LIN {X 0,Y 250.03,Z 323.645,A -85,B 0,C 180,E1 -18844.205,E2 -18844.205} C_VEL
LIN {X 0,Y 249.102,Z 319.461,A -85,B 0,C 180,E1 -18845.837,E2 -18845.837} C_VEL
LIN {X 0,Y 249.003,Z 319.471,A -85,B 0,C 180,E1 -18850.477,E2 -18850.477} C_VEL
LIN {X 0,Y 248.982,Z 319.471,A -85,B 0,C 180,E1 -18854.882,E2 -18854.882} C_VEL
LIN {X 0,Y 249.005,Z 319.467,A -85,B 0,C 180,E1 -18857.361,E2 -18857.361} C_VEL
LIN {X 0,Y 249.035,Z 319.463,A -85,B 0,C 180,E1 -18861.621,E2 -18861.621} C_VEL
LIN {X 0,Y 249.057,Z 319.458,A -85,B 0,C 180,E1 -18865.642,E2 -18865.642} C_VEL
LIN {X 0,Y 249.047,Z 319.447,A -85,B 0,C 180,E1 -18869.473,E2 -18869.473} C_VEL
LIN {X 0,Y 249.068,Z 319.461,A -85,B 0,C 180,E1 -18873.162,E2 -18873.162} C_VEL
LIN {X 0,Y 249.074,Z 319.46,A -85,B 0,C 180,E1 -18876.732,E2 -18876.732} C_VEL
LIN {X 0,Y 249.105,Z 319.45,A -85,B 0,C 180,E1 -18880.211,E2 -18880.211} C_VEL
LIN {X 0,Y 249.237,Z 319.439,A -85,B 0,C 180,E1 -18883.622,E2 -18883.622} C_VEL
LIN {X 0,Y 249.248,Z 319.429,A -85,B 0,C 180,E1 -18888.617,E2 -18888.617} C_VEL
LIN {X 0,Y 249.477,Z 319.408,A -85,B 0,C 180,E1 -18891.903,E2 -18891.903} C_VEL
LIN {X 0,Y 249.43,Z 319.409,A -85,B 0,C 180,E1 -18896.77,E2 -18896.77} C_VEL
LIN {X 0,Y 249.722,Z 319.373,A -85,B 0,C 180,E1 -18900,E2 -18900} C_VEL
LIN {X 0,Y 249.427,Z 319.411,A -85,B 0,C 180,E1 -18903.231,E2 -18903.231} C_VEL
LIN {X 0,Y 249.428,Z 319.41,A -85,B 0,C 180,E1 -18906.549,E2 -18906.549} C_VEL
LIN {X 0,Y 249.339,Z 319.421,A -85,B 0,C 180,E1 -18909.737,E2 -18909.737} C_VEL
LIN {X 0,Y 249.201,Z 319.438,A -85,B 0,C 180,E1 -18914.704,E2 -18914.704} C_VEL
LIN {X 0,Y 249.134,Z 319.451,A -85,B 0,C 180,E1 -18918.078,E2 -18918.078} C_VEL
LIN {X 0,Y 249.079,Z 319.453,A -85,B 0,C 180,E1 -18921.519,E2 -18921.519} C_VEL
LIN {X 0,Y 249.081,Z 319.443,A -85,B 0,C 180,E1 -18925.461,E2 -18925.461} C_VEL
LIN {X 0,Y 249.035,Z 319.46,A -85,B 0,C 180,E1 -18928.976,E2 -18928.976} C_VEL
LIN {X 0,Y 249.024,Z 319.466,A -85,B 0,C 180,E1 -18932.427,E2 -18932.427} C_VEL
LIN {X 0,Y 249.044,Z 319.461,A -85,B 0,C 180,E1 -18936.344,E2 -18936.344} C_VEL
LIN {X 0,Y 249.004,Z 319.457,A -85,B 0,C 180,E1 -18940.479,E2 -18940.479} C_VEL
LIN {X 0,Y 248.984,Z 319.47,A -85,B 0,C 180,E1 -18944.884,E2 -18944.884} C_VEL
LIN {X 0,Y 249,Z 319.467,A -85,B 0,C 180,E1 -18947.361,E2 -18947.361} C_VEL
LIN {X 0,Y 249.041,Z 319.453,A -85,B 0,C 180,E1 -18952.202,E2 -18952.202} C_VEL
LIN {X 0,Y 249.043,Z 319.461,A -85,B 0,C 180,E1 -18955.641,E2 -18955.641} C_VEL
LIN {X 0,Y 249.002,Z 319.468,A -85,B 0,C 180,E1 -18959.468,E2 -18959.468} C_VEL
LIN {X 0,Y 249.036,Z 319.464,A -85,B 0,C 180,E1 -18963.159,E2 -18963.159} C_VEL
LIN {X 0,Y 249.055,Z 319.459,A -85,B 0,C 180,E1 -18966.731,E2 -18966.731} C_VEL
LIN {X 0,Y 249.088,Z 319.455,A -85,B 0,C 180,E1 -18970.211,E2 -18970.211} C_VEL
LIN {X 0,Y 249.198,Z 319.444,A -85,B 0,C 180,E1 -18973.62,E2 -18973.62} C_VEL
LIN {X 0,Y 249.245,Z 319.436,A -85,B 0,C 180,E1 -18978.617,E2 -18978.617} C_VEL
LIN {X 0,Y 249.438,Z 319.415,A -85,B 0,C 180,E1 -18981.902,E2 -18981.902} C_VEL
LIN {X 0,Y 249.255,Z 319.435,A -85,B 0,C 180,E1 -18985.149,E2 -18985.149} C_VEL
LIN {X 0,Y 249.65,Z 319.389,A -85,B 0,C 180,E1 -18988.388,E2 -18988.388} C_VEL
LIN {X 0,Y 249.649,Z 319.388,A -85,B 0,C 180,E1 -18991.614,E2 -18991.614} C_VEL
LIN {X 0,Y 249.424,Z 319.418,A -85,B 0,C 180,E1 -18996.472,E2 -18996.472} C_VEL
LIN {X 0,Y 249.335,Z 319.426,A -85,B 0,C 180,E1 -18999.738,E2 -18999.738} C_VEL
LIN {X 0,Y 249.146,Z 319.452,A -85,B 0,C 180,E1 -19004.708,E2 -19004.708} C_VEL
LIN {X 0,Y 249.137,Z 319.452,A -85,B 0,C 180,E1 -19007.325,E2 -19007.325} C_VEL
LIN {X 0,Y 250.767,Z 323.932,A -85,B 0,C 180,E1 -19007.655,E2 -19007.655} C_VEL
LIN {X 0,Y 258.308,Z 343.81,A -85,B 0,C 180,E1 -19009.057,E2 -19009.057} C_VEL
LIN {X 0,Y 262.117,Z 355.153,A -85,B 0,C 180,E1 -19009.774,E2 -19009.774} C_VEL
LIN {X 0,Y 259.34,Z 426.653,A -85,B 0,C 180,E1 -19012.022,E2 -19012.022} C_VEL
LIN {X 0,Y 258.384,Z 440.539,A -85,B 0,C 180,E1 -19012.778,E2 -19012.778} C_VEL
LIN {X 0,Y 257.341,Z 452.554,A -85,B 0,C 180,E1 -19013.731,E2 -19013.731} C_VEL
LIN {X 0,Y 255.946,Z 464.685,A -85,B 0,C 180,E1 -19015.02,E2 -19015.02} C_VEL
LIN {X 0,Y 254.367,Z 476.702,A -85,B 0,C 180,E1 -19016.671,E2 -19016.671} C_VEL
LIN {X 0,Y 252.928,Z 486.716,A -85,B 0,C 180,E1 -19018.415,E2 -19018.415} C_VEL
LIN {X 0,Y 251.406,Z 496.138,A -85,B 0,C 180,E1 -19020.444,E2 -19020.444} C_VEL
LIN {X 0,Y 250.107,Z 504.061,A -85,B 0,C 180,E1 -19022.541,E2 -19022.541} C_VEL
LIN {X 0,Y 248.917,Z 511.656,A -85,B 0,C 180,E1 -19025.034,E2 -19025.034} C_VEL
LIN {X 0,Y 248.031,Z 517.544,A -85,B 0,C 180,E1 -19027.496,E2 -19027.496} C_VEL
LIN {X 0,Y 247.458,Z 522.104,A -85,B 0,C 180,E1 -19029.93,E2 -19029.93} C_VEL
LIN {X 0,Y 246.793,Z 526.425,A -85,B 0,C 180,E1 -19033.115,E2 -19033.115} C_VEL
LIN {X 0,Y 246.614,Z 528.472,A -85,B 0,C 180,E1 -19035.435,E2 -19035.435} C_VEL
LIN {X 0,Y 246.681,Z 529.69,A -85,B 0,C 180,E1 -19037.796,E2 -19037.796} C_VEL
LIN {X 0,Y 246.872,Z 530.061,A -85,B 0,C 180,E1 -19040.233,E2 -19040.233} C_VEL
LIN {X 0,Y 247.505,Z 529.204,A -85,B 0,C 180,E1 -19043.394,E2 -19043.394} C_VEL
LIN {X 0,Y 248.58,Z 526.802,A -85,B 0,C 180,E1 -19046.542,E2 -19046.542} C_VEL
LIN {X 0,Y 250.07,Z 522.874,A -85,B 0,C 180,E1 -19049.61,E2 -19049.61} C_VEL
LIN {X 0,Y 251.955,Z 517.798,A -85,B 0,C 180,E1 -19052.381,E2 -19052.381} C_VEL
LIN {X 0,Y 254.299,Z 511.152,A -85,B 0,C 180,E1 -19055.073,E2 -19055.073} C_VEL
LIN {X 0,Y 256.78,Z 503.593,A -85,B 0,C 180,E1 -19057.469,E2 -19057.469} C_VEL
LIN {X 0,Y 259.517,Z 494.561,A -85,B 0,C 180,E1 -19059.713,E2 -19059.713} C_VEL
LIN {X 0,Y 262.243,Z 484.71,A -85,B 0,C 180,E1 -19061.645,E2 -19061.645} C_VEL
LIN {X 0,Y 264.805,Z 474.366,A -85,B 0,C 180,E1 -19063.258,E2 -19063.258} C_VEL
LIN {X 0,Y 267.225,Z 462.907,A -85,B 0,C 180,E1 -19064.654,E2 -19064.654} C_VEL
LIN {X 0,Y 269.363,Z 450.034,A -85,B 0,C 180,E1 -19065.862,E2 -19065.862} C_VEL
LIN {X 0,Y 270.921,Z 437.319,A -85,B 0,C 180,E1 -19066.734,E2 -19066.734} C_VEL
LIN {X 0,Y 272.145,Z 423.426,A -85,B 0,C 180,E1 -19067.343,E2 -19067.343} C_VEL
LIN {X 0,Y 275.677,Z 365.669,A -85,B 0,C 180,E1 -19069.121,E2 -19069.121} C_VEL
LIN {X 0,Y 270.019,Z 353.323,A -85,B 0,C 180,E1 -19070.753,E2 -19070.753} C_VEL
LIN {X 0,Y 263.673,Z 341.842,A -85,B 0,C 180,E1 -19072.672,E2 -19072.672} C_VEL
LIN {X 0,Y 259.384,Z 334.783,A -85,B 0,C 180,E1 -19074.07,E2 -19074.07} C_VEL
LIN {X 0,Y 256.653,Z 330.712,A -85,B 0,C 180,E1 -19074.992,E2 -19074.992} C_VEL
LIN {X 0,Y 250.933,Z 322.884,A -85,B 0,C 180,E1 -19077.065,E2 -19077.065} C_VEL
LIN {X 0,Y 249.681,Z 321.815,A -85,B 0,C 180,E1 -19077.526,E2 -19077.526} C_VEL
LIN {X 0,Y 248.305,Z 321.348,A -85,B 0,C 180,E1 -19078.029,E2 -19078.029} C_VEL
LIN {X 0,Y 244.436,Z 320.951,A -85,B 0,C 180,E1 -19079.7,E2 -19079.7} C_VEL
LIN {X 0,Y 242.856,Z 320.376,A -85,B 0,C 180,E1 -19080.934,E2 -19080.934} C_VEL
LIN {X 0,Y 242.635,Z 320.256,A -85,B 0,C 180,E1 -19081.579,E2 -19081.579} C_VEL
LIN {X 0,Y 242.411,Z 320.281,A -85,B 0,C 180,E1 -19086.659,E2 -19086.659} C_VEL
LIN {X 0,Y 242.27,Z 320.297,A -85,B 0,C 180,E1 -19090.023,E2 -19090.023} C_VEL
LIN {X 0,Y 242.139,Z 320.323,A -85,B 0,C 180,E1 -19095.142,E2 -19095.142} C_VEL
LIN {X 0,Y 242.052,Z 320.331,A -85,B 0,C 180,E1 -19098.625,E2 -19098.625} C_VEL
LIN {X 0,Y 242.007,Z 320.335,A -85,B 0,C 180,E1 -19102.18,E2 -19102.18} C_VEL
LIN {X 0,Y 242.069,Z 320.328,A -85,B 0,C 180,E1 -19105.838,E2 -19105.838} C_VEL
LIN {X 0,Y 242.031,Z 320.336,A -85,B 0,C 180,E1 -19109.58,E2 -19109.58} C_VEL
LIN {X 0,Y 241.983,Z 320.342,A -85,B 0,C 180,E1 -19113.492,E2 -19113.492} C_VEL
LIN {X 0,Y 241.991,Z 320.335,A -85,B 0,C 180,E1 -19117.581,E2 -19117.581} C_VEL
LIN {X 0,Y 241.971,Z 320.532,A -85,B 0,C 180,E1 -19121.083,E2 -19121.083} C_VEL
LIN {X 0,Y 243.323,Z 324.398,A -85,B 0,C 180,E1 -19123.884,E2 -19123.884} C_VEL
LIN {X 0,Y 245.036,Z 329.254,A -85,B 0,C 180,E1 -19127.001,E2 -19127.001} C_VEL
LIN {X 0,Y 245.857,Z 331.663,A -85,B 0,C 180,E1 -19128.294,E2 -19128.294} C_VEL
LIN {X 0,Y 249.084,Z 336.698,A -85,B 0,C 180,E1 -19129.624,E2 -19129.624} C_VEL
LIN {X 0,Y 253.954,Z 344.732,A -85,B 0,C 180,E1 -19131.478,E2 -19131.478} C_VEL
LIN {X 0,Y 257.084,Z 350.374,A -85,B 0,C 180,E1 -19132.593,E2 -19132.593} C_VEL
LIN {X 0,Y 261.696,Z 359.399,A -85,B 0,C 180,E1 -19134.165,E2 -19134.165} C_VEL
LIN {X 0,Y 266.799,Z 370.947,A -85,B 0,C 180,E1 -19135.818,E2 -19135.818} C_VEL
LIN {X 0,Y 268.746,Z 386.31,A -85,B 0,C 180,E1 -19136.893,E2 -19136.893} C_VEL
LIN {X 0,Y 269.128,Z 390.539,A -85,B 0,C 180,E1 -19137.149,E2 -19137.149} C_VEL
LIN {X 0,Y 265.736,Z 443.432,A -85,B 0,C 180,E1 -19138.843,E2 -19138.843} C_VEL
LIN {X 0,Y 264.156,Z 456.738,A -85,B 0,C 180,E1 -19139.524,E2 -19139.524} C_VEL
LIN {X 0,Y 261.95,Z 469.593,A -85,B 0,C 180,E1 -19140.462,E2 -19140.462} C_VEL
LIN {X 0,Y 259.418,Z 481.764,A -85,B 0,C 180,E1 -19141.698,E2 -19141.698} C_VEL
LIN {X 0,Y 256.562,Z 492.835,A -85,B 0,C 180,E1 -19143.128,E2 -19143.128} C_VEL
LIN {X 0,Y 253.881,Z 502.949,A -85,B 0,C 180,E1 -19144.81,E2 -19144.81} C_VEL
LIN {X 0,Y 251.337,Z 511.329,A -85,B 0,C 180,E1 -19146.517,E2 -19146.517} C_VEL
LIN {X 0,Y 248.356,Z 520.484,A -85,B 0,C 180,E1 -19148.85,E2 -19148.85} C_VEL
LIN {X 0,Y 245.962,Z 527.909,A -85,B 0,C 180,E1 -19151.248,E2 -19151.248} C_VEL
LIN {X 0,Y 243.566,Z 534.796,A -85,B 0,C 180,E1 -19154.09,E2 -19154.09} C_VEL
LIN {X 0,Y 241.883,Z 539.395,A -85,B 0,C 180,E1 -19156.558,E2 -19156.558} C_VEL
LIN {X 0,Y 240.875,Z 542.931,A -85,B 0,C 180,E1 -19159.067,E2 -19159.067} C_VEL
LIN {X 0,Y 240.207,Z 545.478,A -85,B 0,C 180,E1 -19161.587,E2 -19161.587} C_VEL
LIN {X 0,Y 239.84,Z 547.387,A -85,B 0,C 180,E1 -19164.956,E2 -19164.956} C_VEL
LIN {X 0,Y 239.816,Z 547.753,A -85,B 0,C 180,E1 -19166.639,E2 -19166.639} C_VEL
LIN {X 0,Y 239.905,Z 547.721,A -85,B 0,C 180,E1 -19168.32,E2 -19168.32} C_VEL
LIN {X 0,Y 239.958,Z 547.237,A -85,B 0,C 180,E1 -19169.999,E2 -19169.999} C_VEL
LIN {X 0,Y 239.945,Z 546.336,A -85,B 0,C 180,E1 -19171.677,E2 -19171.677} C_VEL
LIN {X 0,Y 239.905,Z 545.015,A -85,B 0,C 180,E1 -19173.358,E2 -19173.358} C_VEL
LIN {X 0,Y 239.916,Z 542.156,A -85,B 0,C 180,E1 -19175.883,E2 -19175.883} C_VEL
LIN {X 0,Y 240.201,Z 538.208,A -85,B 0,C 180,E1 -19178.411,E2 -19178.411} C_VEL
LIN {X 0,Y 240.846,Z 532.063,A -85,B 0,C 180,E1 -19181.359,E2 -19181.359} C_VEL
LIN {X 0,Y 241.813,Z 525.276,A -85,B 0,C 180,E1 -19183.872,E2 -19183.872} C_VEL
LIN {X 0,Y 243.178,Z 516.827,A -85,B 0,C 180,E1 -19186.365,E2 -19186.365} C_VEL
LIN {X 0,Y 244.719,Z 507.213,A -85,B 0,C 180,E1 -19188.61,E2 -19188.61} C_VEL
LIN {X 0,Y 246.198,Z 497.332,A -85,B 0,C 180,E1 -19190.467,E2 -19190.467} C_VEL
LIN {X 0,Y 247.876,Z 486.712,A -85,B 0,C 180,E1 -19192.065,E2 -19192.065} C_VEL
LIN {X 0,Y 249.528,Z 474.972,A -85,B 0,C 180,E1 -19193.442,E2 -19193.442} C_VEL
LIN {X 0,Y 250.995,Z 461.662,A -85,B 0,C 180,E1 -19194.613,E2 -19194.613} C_VEL
LIN {X 0,Y 252.092,Z 449.229,A -85,B 0,C 180,E1 -19195.38,E2 -19195.38} C_VEL
LIN {X 0,Y 252.828,Z 433.94,A -85,B 0,C 180,E1 -19195.963,E2 -19195.963} C_VEL
LIN {X 0,Y 254.548,Z 385.732,A -85,B 0,C 180,E1 -19197.51,E2 -19197.51} C_VEL
LIN {X 0,Y 249.883,Z 349.342,A -85,B 0,C 180,E1 -19199.23,E2 -19199.23} C_VEL
LIN {X 0,Y 245.337,Z 336.056,A -85,B 0,C 180,E1 -19200.196,E2 -19200.196} C_VEL
LIN {X 0,Y 243.169,Z 325.344,A -85,B 0,C 180,E1 -19204.302,E2 -19204.302} C_VEL
LIN {X 0,Y 242.085,Z 320.336,A -85,B 0,C 180,E1 -19206.34,E2 -19206.34} C_VEL
LIN {X 0,Y 241.928,Z 320.349,A -85,B 0,C 180,E1 -19210.949,E2 -19210.949} C_VEL
LIN {X 0,Y 241.915,Z 320.352,A -85,B 0,C 180,E1 -19214.204,E2 -19214.204} C_VEL
LIN {X 0,Y 241.935,Z 320.349,A -85,B 0,C 180,E1 -19218.077,E2 -19218.077} C_VEL
LIN {X 0,Y 241.999,Z 320.342,A -85,B 0,C 180,E1 -19222.42,E2 -19222.42} C_VEL
LIN {X 0,Y 241.987,Z 320.341,A -85,B 0,C 180,E1 -19226.509,E2 -19226.509} C_VEL
LIN {X 0,Y 242.032,Z 320.322,A -85,B 0,C 180,E1 -19230.587,E2 -19230.587} C_VEL
LIN {X 0,Y 242.063,Z 320.331,A -85,B 0,C 180,E1 -19234.183,E2 -19234.183} C_VEL
LIN {X 0,Y 242.048,Z 320.331,A -85,B 0,C 180,E1 -19238.297,E2 -19238.297} C_VEL
LIN {X 0,Y 242.158,Z 320.323,A -85,B 0,C 180,E1 -19243.278,E2 -19243.278} C_VEL
LIN {X 0,Y 242.181,Z 320.309,A -85,B 0,C 180,E1 -19248.28,E2 -19248.28} C_VEL
LIN {X 0,Y 242.423,Z 320.288,A -85,B 0,C 180,E1 -19251.666,E2 -19251.666} C_VEL
LIN {X 0,Y 242.254,Z 320.306,A -85,B 0,C 180,E1 -19255.007,E2 -19255.007} C_VEL
LIN {X 0,Y 242.631,Z 320.251,A -85,B 0,C 180,E1 -19258.341,E2 -19258.341} C_VEL
LIN {X 0,Y 242.63,Z 320.257,A -85,B 0,C 180,E1 -19261.66,E2 -19261.66} C_VEL
LIN {X 0,Y 242.404,Z 320.285,A -85,B 0,C 180,E1 -19266.66,E2 -19266.66} C_VEL
LIN {X 0,Y 242.263,Z 320.298,A -85,B 0,C 180,E1 -19270.024,E2 -19270.024} C_VEL
LIN {X 0,Y 242.163,Z 320.313,A -85,B 0,C 180,E1 -19275.142,E2 -19275.142} C_VEL
LIN {X 0,Y 242.068,Z 320.329,A -85,B 0,C 180,E1 -19278.625,E2 -19278.625} C_VEL
LIN {X 0,Y 242.001,Z 320.336,A -85,B 0,C 180,E1 -19282.182,E2 -19282.182} C_VEL
LIN {X 0,Y 242.029,Z 320.321,A -85,B 0,C 180,E1 -19285.822,E2 -19285.822} C_VEL
LIN {X 0,Y 241.966,Z 320.339,A -85,B 0,C 180,E1 -19289.589,E2 -19289.589} C_VEL
LIN {X 0,Y 241.976,Z 320.341,A -85,B 0,C 180,E1 -19293.494,E2 -19293.494} C_VEL
LIN {X 0,Y 241.986,Z 320.334,A -85,B 0,C 180,E1 -19297.583,E2 -19297.583} C_VEL
LIN {X 0,Y 241.931,Z 320.34,A -85,B 0,C 180,E1 -19301.924,E2 -19301.924} C_VEL
LIN {X 0,Y 241.919,Z 320.349,A -85,B 0,C 180,E1 -19306.576,E2 -19306.576} C_VEL
LIN {X 0,Y 241.992,Z 320.332,A -85,B 0,C 180,E1 -19311.642,E2 -19311.642} C_VEL
LIN {X 0,Y 241.986,Z 320.335,A -85,B 0,C 180,E1 -19314.491,E2 -19314.491} C_VEL
LIN {X 0,Y 241.953,Z 320.344,A -85,B 0,C 180,E1 -19318.478,E2 -19318.478} C_VEL
LIN {X 0,Y 241.968,Z 320.342,A -85,B 0,C 180,E1 -19322.309,E2 -19322.309} C_VEL
LIN {X 0,Y 242.026,Z 320.336,A -85,B 0,C 180,E1 -19326.014,E2 -19326.014} C_VEL
LIN {X 0,Y 242.023,Z 320.338,A -85,B 0,C 180,E1 -19329.608,E2 -19329.608} C_VEL
LIN {X 0,Y 242.118,Z 320.324,A -85,B 0,C 180,E1 -19333.317,E2 -19333.317} C_VEL
LIN {X 0,Y 242.156,Z 320.318,A -85,B 0,C 180,E1 -19336.576,E2 -19336.576} C_VEL
LIN {X 0,Y 242.388,Z 320.291,A -85,B 0,C 180,E1 -19341.665,E2 -19341.665} C_VEL
LIN {X 0,Y 242.403,Z 320.289,A -85,B 0,C 180,E1 -19343.341,E2 -19343.341} C_VEL
LIN {X 0,Y 242.609,Z 320.266,A -85,B 0,C 180,E1 -19348.341,E2 -19348.341} C_VEL
LIN {X 0,Y 242.609,Z 320.265,A -85,B 0,C 180,E1 -19351.661,E2 -19351.661} C_VEL
LIN {X 0,Y 242.394,Z 320.293,A -85,B 0,C 180,E1 -19356.661,E2 -19356.661} C_VEL
LIN {X 0,Y 242.263,Z 320.308,A -85,B 0,C 180,E1 -19360.025,E2 -19360.025} C_VEL
LIN {X 0,Y 242.105,Z 320.329,A -85,B 0,C 180,E1 -19365.146,E2 -19365.146} C_VEL
LIN {X 0,Y 242.124,Z 320.327,A -85,B 0,C 180,E1 -19366.651,E2 -19366.651} C_VEL
LIN {X 0,Y 243.549,Z 324.322,A -85,B 0,C 180,E1 -19366.962,E2 -19366.962} C_VEL
LIN {X 0,Y 248.831,Z 337.497,A -85,B 0,C 180,E1 -19367.96,E2 -19367.96} C_VEL
LIN {X 0,Y 255.38,Z 356.241,A -85,B 0,C 180,E1 -19369.232,E2 -19369.232} C_VEL
LIN {X 0,Y 252.609,Z 426.976,A -85,B 0,C 180,E1 -19371.525,E2 -19371.525} C_VEL
LIN {X 0,Y 251.648,Z 440.232,A -85,B 0,C 180,E1 -19372.258,E2 -19372.258} C_VEL
LIN {X 0,Y 250.597,Z 452.306,A -85,B 0,C 180,E1 -19373.228,E2 -19373.228} C_VEL
LIN {X 0,Y 249.119,Z 464.887,A -85,B 0,C 180,E1 -19374.591,E2 -19374.591} C_VEL
LIN {X 0,Y 247.486,Z 476.854,A -85,B 0,C 180,E1 -19376.274,E2 -19376.274} C_VEL
LIN {X 0,Y 245.91,Z 487.572,A -85,B 0,C 180,E1 -19378.203,E2 -19378.203} C_VEL
LIN {X 0,Y 244.314,Z 497.132,A -85,B 0,C 180,E1 -19380.345,E2 -19380.345} C_VEL
LIN {X 0,Y 243.082,Z 504.382,A -85,B 0,C 180,E1 -19382.336,E2 -19382.336} C_VEL
LIN {X 0,Y 241.834,Z 512.047,A -85,B 0,C 180,E1 -19384.933,E2 -19384.933} C_VEL
LIN {X 0,Y 240.877,Z 518.544,A -85,B 0,C 180,E1 -19387.787,E2 -19387.787} C_VEL
LIN {X 0,Y 240.219,Z 523.22,A -85,B 0,C 180,E1 -19390.476,E2 -19390.476} C_VEL
LIN {X 0,Y 239.73,Z 526.314,A -85,B 0,C 180,E1 -19392.868,E2 -19392.868} C_VEL
LIN {X 0,Y 239.532,Z 528.483,A -85,B 0,C 180,E1 -19395.236,E2 -19395.236} C_VEL
LIN {X 0,Y 239.591,Z 529.814,A -85,B 0,C 180,E1 -19397.571,E2 -19397.571} C_VEL
LIN {X 0,Y 239.748,Z 530.34,A -85,B 0,C 180,E1 -19399.84,E2 -19399.84} C_VEL
LIN {X 0,Y 240.119,Z 530.09,A -85,B 0,C 180,E1 -19402.211,E2 -19402.211} C_VEL
LIN {X 0,Y 240.827,Z 528.903,A -85,B 0,C 180,E1 -19404.798,E2 -19404.798} C_VEL
LIN {X 0,Y 241.866,Z 526.68,A -85,B 0,C 180,E1 -19407.424,E2 -19407.424} C_VEL
LIN {X 0,Y 243.251,Z 523.312,A -85,B 0,C 180,E1 -19410.085,E2 -19410.085} C_VEL
LIN {X 0,Y 245.101,Z 518.698,A -85,B 0,C 180,E1 -19412.735,E2 -19412.735} C_VEL
LIN {X 0,Y 247.418,Z 512.645,A -85,B 0,C 180,E1 -19415.365,E2 -19415.365} C_VEL
LIN {X 0,Y 250.163,Z 504.78,A -85,B 0,C 180,E1 -19417.987,E2 -19417.987} C_VEL
LIN {X 0,Y 253.136,Z 495.698,A -85,B 0,C 180,E1 -19420.349,E2 -19420.349} C_VEL
LIN {X 0,Y 255.77,Z 486.696,A -85,B 0,C 180,E1 -19422.2,E2 -19422.2} C_VEL
LIN {X 0,Y 258.828,Z 475.208,A -85,B 0,C 180,E1 -19424.072,E2 -19424.072} C_VEL
LIN {X 0,Y 261.347,Z 464.019,A -85,B 0,C 180,E1 -19425.49,E2 -19425.49} C_VEL
LIN {X 0,Y 263.611,Z 451.481,A -85,B 0,C 180,E1 -19426.706,E2 -19426.706} C_VEL
LIN {X 0,Y 265.308,Z 438.816,A -85,B 0,C 180,E1 -19427.619,E2 -19427.619} C_VEL
LIN {X 0,Y 266.587,Z 425.001,A -85,B 0,C 180,E1 -19428.264,E2 -19428.264} C_VEL
LIN {X 0,Y 270.177,Z 367.755,A -85,B 0,C 180,E1 -19430.076,E2 -19430.076} C_VEL
LIN {X 0,Y 264.553,Z 355.604,A -85,B 0,C 180,E1 -19431.817,E2 -19431.817} C_VEL
LIN {X 0,Y 258.185,Z 344.023,A -85,B 0,C 180,E1 -19433.896,E2 -19433.896} C_VEL
LIN {X 0,Y 253.236,Z 336.294,A -85,B 0,C 180,E1 -19435.617,E2 -19435.617} C_VEL
LIN {X 0,Y 245.251,Z 324.921,A -85,B 0,C 180,E1 -19438.773,E2 -19438.773} C_VEL
LIN {X 0,Y 243.331,Z 322.513,A -85,B 0,C 180,E1 -19439.601,E2 -19439.601} C_VEL
LIN {X 0,Y 243.054,Z 321.797,A -85,B 0,C 180,E1 -19439.772,E2 -19439.772} C_VEL
LIN {X 0,Y 242.628,Z 320.256,A -85,B 0,C 180,E1 -19440.933,E2 -19440.933} C_VEL
LIN {X 0,Y 242.635,Z 320.256,A -85,B 0,C 180,E1 -19441.579,E2 -19441.579} C_VEL
LIN {X 0,Y 242.34,Z 320.299,A -85,B 0,C 180,E1 -19442.504,E2 -19442.504} C_VEL
LIN {X 0,Y 240.983,Z 320.474,A -85,B 0,C 180,E1 -19443.867,E2 -19443.867} C_VEL
LIN {X 0,Y 236.525,Z 321.032,A -85,B 0,C 180,E1 -19447.045,E2 -19447.045} C_VEL
LIN {X 0,Y 235.408,Z 321.162,A -85,B 0,C 180,E1 -19448.471,E2 -19448.471} C_VEL
LIN {X 0,Y 235.303,Z 321.171,A -85,B 0,C 180,E1 -19448.955,E2 -19448.955} C_VEL
LIN {X 0,Y 235.093,Z 321.19,A -85,B 0,C 180,E1 -19453.836,E2 -19453.836} C_VEL
LIN {X 0,Y 235.021,Z 321.199,A -85,B 0,C 180,E1 -19457.399,E2 -19457.399} C_VEL
LIN {X 0,Y 234.978,Z 321.209,A -85,B 0,C 180,E1 -19461.998,E2 -19461.998} C_VEL
LIN {X 0,Y 234.971,Z 321.212,A -85,B 0,C 180,E1 -19466.657,E2 -19466.657} C_VEL
LIN {X 0,Y 234.933,Z 321.214,A -85,B 0,C 180,E1 -19470.567,E2 -19470.567} C_VEL
LIN {X 0,Y 234.932,Z 321.212,A -85,B 0,C 180,E1 -19474.637,E2 -19474.637} C_VEL
LIN {X 0,Y 234.969,Z 321.317,A -85,B 0,C 180,E1 -19478.226,E2 -19478.226} C_VEL
LIN {X 0,Y 237.053,Z 327.105,A -85,B 0,C 180,E1 -19482.991,E2 -19482.991} C_VEL
LIN {X 0,Y 238.301,Z 330.865,A -85,B 0,C 180,E1 -19485.507,E2 -19485.507} C_VEL
LIN {X 0,Y 242.379,Z 336.87,A -85,B 0,C 180,E1 -19487.449,E2 -19487.449} C_VEL
LIN {X 0,Y 246.9,Z 344.12,A -85,B 0,C 180,E1 -19489.396,E2 -19489.396} C_VEL
LIN {X 0,Y 251,Z 351.189,A -85,B 0,C 180,E1 -19491.025,E2 -19491.025} C_VEL
LIN {X 0,Y 255.403,Z 359.563,A -85,B 0,C 180,E1 -19492.644,E2 -19492.644} C_VEL
LIN {X 0,Y 260,Z 369.572,A -85,B 0,C 180,E1 -19494.269,E2 -19494.269} C_VEL
LIN {X 0,Y 262.019,Z 374.909,A -85,B 0,C 180,E1 -19494.975,E2 -19494.975} C_VEL
LIN {X 0,Y 263.585,Z 388.526,A -85,B 0,C 180,E1 -19495.949,E2 -19495.949} C_VEL
LIN {X 0,Y 263.739,Z 393.029,A -85,B 0,C 180,E1 -19496.189,E2 -19496.189} C_VEL
LIN {X 0,Y 260.34,Z 443.254,A -85,B 0,C 180,E1 -19497.837,E2 -19497.837} C_VEL
LIN {X 0,Y 258.671,Z 456.525,A -85,B 0,C 180,E1 -19498.521,E2 -19498.521} C_VEL
LIN {X 0,Y 256.509,Z 468.848,A -85,B 0,C 180,E1 -19499.429,E2 -19499.429} C_VEL
LIN {X 0,Y 254.017,Z 480.361,A -85,B 0,C 180,E1 -19500.586,E2 -19500.586} C_VEL
LIN {X 0,Y 250.689,Z 492.897,A -85,B 0,C 180,E1 -19502.219,E2 -19502.219} C_VEL
LIN {X 0,Y 247.835,Z 502.895,A -85,B 0,C 180,E1 -19503.924,E2 -19503.924} C_VEL
LIN {X 0,Y 244.893,Z 512.008,A -85,B 0,C 180,E1 -19505.86,E2 -19505.86} C_VEL
LIN {X 0,Y 241.738,Z 521.119,A -85,B 0,C 180,E1 -19508.287,E2 -19508.287} C_VEL
LIN {X 0,Y 239.245,Z 528.295,A -85,B 0,C 180,E1 -19510.708,E2 -19510.708} C_VEL
LIN {X 0,Y 236.739,Z 534.99,A -85,B 0,C 180,E1 -19513.618,E2 -19513.618} C_VEL
LIN {X 0,Y 234.955,Z 539.477,A -85,B 0,C 180,E1 -19516.154,E2 -19516.154} C_VEL
LIN {X 0,Y 234.222,Z 541.87,A -85,B 0,C 180,E1 -19517.874,E2 -19517.874} C_VEL
LIN {X 0,Y 233.597,Z 543.84,A -85,B 0,C 180,E1 -19519.599,E2 -19519.599} C_VEL
LIN {X 0,Y 233.177,Z 545.357,A -85,B 0,C 180,E1 -19521.331,E2 -19521.331} C_VEL
LIN {X 0,Y 232.743,Z 547.179,A -85,B 0,C 180,E1 -19524.802,E2 -19524.802} C_VEL
LIN {X 0,Y 232.72,Z 547.503,A -85,B 0,C 180,E1 -19526.536,E2 -19526.536} C_VEL
LIN {X 0,Y 232.812,Z 547.391,A -85,B 0,C 180,E1 -19528.269,E2 -19528.269} C_VEL
LIN {X 0,Y 232.888,Z 546.858,A -85,B 0,C 180,E1 -19529.999,E2 -19529.999} C_VEL
LIN {X 0,Y 232.876,Z 545.913,A -85,B 0,C 180,E1 -19531.728,E2 -19531.728} C_VEL
LIN {X 0,Y 232.807,Z 544.544,A -85,B 0,C 180,E1 -19533.46,E2 -19533.46} C_VEL
LIN {X 0,Y 232.855,Z 541.599,A -85,B 0,C 180,E1 -19536.063,E2 -19536.063} C_VEL
LIN {X 0,Y 233.164,Z 537.556,A -85,B 0,C 180,E1 -19538.667,E2 -19538.667} C_VEL
LIN {X 0,Y 233.845,Z 531.257,A -85,B 0,C 180,E1 -19541.703,E2 -19541.703} C_VEL
LIN {X 0,Y 234.899,Z 524.358,A -85,B 0,C 180,E1 -19544.289,E2 -19544.289} C_VEL
LIN {X 0,Y 236.351,Z 515.734,A -85,B 0,C 180,E1 -19546.852,E2 -19546.852} C_VEL
LIN {X 0,Y 237.811,Z 506.82,A -85,B 0,C 180,E1 -19548.969,E2 -19548.969} C_VEL
LIN {X 0,Y 239.529,Z 495.851,A -85,B 0,C 180,E1 -19551.064,E2 -19551.064} C_VEL
LIN {X 0,Y 241.193,Z 484.865,A -85,B 0,C 180,E1 -19552.71,E2 -19552.71} C_VEL
LIN {X 0,Y 243.037,Z 472.734,A -85,B 0,C 180,E1 -19554.107,E2 -19554.107} C_VEL
LIN {X 0,Y 244.252,Z 461.383,A -85,B 0,C 180,E1 -19555.112,E2 -19555.112} C_VEL
LIN {X 0,Y 245.372,Z 448.971,A -85,B 0,C 180,E1 -19555.898,E2 -19555.898} C_VEL
LIN {X 0,Y 246.121,Z 433.789,A -85,B 0,C 180,E1 -19556.497,E2 -19556.497} C_VEL
LIN {X 0,Y 247.891,Z 386.332,A -85,B 0,C 180,E1 -19558.064,E2 -19558.064} C_VEL
LIN {X 0,Y 243.343,Z 351.084,A -85,B 0,C 180,E1 -19559.777,E2 -19559.777} C_VEL
LIN {X 0,Y 238.08,Z 335.915,A -85,B 0,C 180,E1 -19560.89,E2 -19560.89} C_VEL
LIN {X 0,Y 235.955,Z 325.599,A -85,B 0,C 180,E1 -19564.984,E2 -19564.984} C_VEL
LIN {X 0,Y 234.998,Z 321.218,A -85,B 0,C 180,E1 -19566.868,E2 -19566.868} C_VEL
LIN {X 0,Y 234.877,Z 321.227,A -85,B 0,C 180,E1 -19571.578,E2 -19571.578} C_VEL
LIN {X 0,Y 234.88,Z 321.226,A -85,B 0,C 180,E1 -19575.898,E2 -19575.898} C_VEL
LIN {X 0,Y 234.891,Z 321.228,A -85,B 0,C 180,E1 -19578.834,E2 -19578.834} C_VEL
LIN {X 0,Y 234.951,Z 321.219,A -85,B 0,C 180,E1 -19581.085,E2 -19581.085} C_VEL
LIN {X 0,Y 234.956,Z 321.216,A -85,B 0,C 180,E1 -19585.367,E2 -19585.367} C_VEL
LIN {X 0,Y 234.965,Z 321.199,A -85,B 0,C 180,E1 -19590.157,E2 -19590.157} C_VEL
LIN {X 0,Y 234.989,Z 321.212,A -85,B 0,C 180,E1 -19593.793,E2 -19593.793} C_VEL
LIN {X 0,Y 235.007,Z 321.21,A -85,B 0,C 180,E1 -19598.97,E2 -19598.97} C_VEL
LIN {X 0,Y 235.092,Z 321.202,A -85,B 0,C 180,E1 -19603.059,E2 -19603.059} C_VEL
LIN {X 0,Y 235.142,Z 321.186,A -85,B 0,C 180,E1 -19607.924,E2 -19607.924} C_VEL
LIN {X 0,Y 235.372,Z 321.165,A -85,B 0,C 180,E1 -19611.414,E2 -19611.414} C_VEL
LIN {X 0,Y 235.399,Z 321.162,A -85,B 0,C 180,E1 -19613.142,E2 -19613.142} C_VEL
LIN {X 0,Y 235.591,Z 321.127,A -85,B 0,C 180,E1 -19618.291,E2 -19618.291} C_VEL
LIN {X 0,Y 235.59,Z 321.134,A -85,B 0,C 180,E1 -19621.71,E2 -19621.71} C_VEL
LIN {X 0,Y 235.355,Z 321.163,A -85,B 0,C 180,E1 -19626.861,E2 -19626.861} C_VEL
LIN {X 0,Y 235.21,Z 321.174,A -85,B 0,C 180,E1 -19630.328,E2 -19630.328} C_VEL
LIN {X 0,Y 235.11,Z 321.192,A -85,B 0,C 180,E1 -19635.607,E2 -19635.607} C_VEL
LIN {X 0,Y 235.003,Z 321.207,A -85,B 0,C 180,E1 -19639.207,E2 -19639.207} C_VEL
LIN {X 0,Y 234.943,Z 321.21,A -85,B 0,C 180,E1 -19642.885,E2 -19642.885} C_VEL
LIN {X 0,Y 234.942,Z 321.209,A -85,B 0,C 180,E1 -19646.661,E2 -19646.661} C_VEL
LIN {X 0,Y 234.896,Z 321.225,A -85,B 0,C 180,E1 -19650.574,E2 -19650.574} C_VEL
LIN {X 0,Y 234.927,Z 321.222,A -85,B 0,C 180,E1 -19654.639,E2 -19654.639} C_VEL
LIN {X 0,Y 234.94,Z 321.208,A -85,B 0,C 180,E1 -19658.946,E2 -19658.946} C_VEL
LIN {X 0,Y 234.876,Z 321.224,A -85,B 0,C 180,E1 -19663.489,E2 -19663.489} C_VEL
LIN {X 0,Y 234.872,Z 321.227,A -85,B 0,C 180,E1 -19666.512,E2 -19666.512} C_VEL
LIN {X 0,Y 234.917,Z 321.217,A -85,B 0,C 180,E1 -19671.08,E2 -19671.08} C_VEL
LIN {X 0,Y 234.929,Z 321.22,A -85,B 0,C 180,E1 -19675.363,E2 -19675.363} C_VEL
LIN {X 0,Y 234.899,Z 321.225,A -85,B 0,C 180,E1 -19679.429,E2 -19679.429} C_VEL
LIN {X 0,Y 234.97,Z 321.215,A -85,B 0,C 180,E1 -19683.808,E2 -19683.808} C_VEL
LIN {X 0,Y 234.991,Z 321.211,A -85,B 0,C 180,E1 -19688.969,E2 -19688.969} C_VEL
LIN {X 0,Y 235.058,Z 321.203,A -85,B 0,C 180,E1 -19693.093,E2 -19693.093} C_VEL
LIN {X 0,Y 235.112,Z 321.199,A -85,B 0,C 180,E1 -19697.923,E2 -19697.923} C_VEL
LIN {X 0,Y 235.322,Z 321.17,A -85,B 0,C 180,E1 -19701.413,E2 -19701.413} C_VEL
LIN {X 0,Y 235.355,Z 321.166,A -85,B 0,C 180,E1 -19703.141,E2 -19703.141} C_VEL
LIN {X 0,Y 235.568,Z 321.144,A -85,B 0,C 180,E1 -19708.291,E2 -19708.291} C_VEL
LIN {X 0,Y 235.567,Z 321.143,A -85,B 0,C 180,E1 -19711.711,E2 -19711.711} C_VEL
LIN {X 0,Y 235.345,Z 321.17,A -85,B 0,C 180,E1 -19716.861,E2 -19716.861} C_VEL
LIN {X 0,Y 235.187,Z 321.19,A -85,B 0,C 180,E1 -19720.33,E2 -19720.33} C_VEL
LIN {X 0,Y 235.046,Z 321.208,A -85,B 0,C 180,E1 -19725.612,E2 -19725.612} C_VEL
LIN {X 0,Y 235.085,Z 321.322,A -85,B 0,C 180,E1 -19725.976,E2 -19725.976} C_VEL
LIN {X 0,Y 236.012,Z 323.987,A -85,B 0,C 180,E1 -19726.178,E2 -19726.178} C_VEL
LIN {X 0,Y 241.767,Z 337.895,A -85,B 0,C 180,E1 -19727.302,E2 -19727.302} C_VEL
LIN {X 0,Y 248.803,Z 357.945,A -85,B 0,C 180,E1 -19728.705,E2 -19728.705} C_VEL
LIN {X 0,Y 245.905,Z 427.111,A -85,B 0,C 180,E1 -19731.006,E2 -19731.006} C_VEL
LIN {X 0,Y 244.849,Z 441.043,A -85,B 0,C 180,E1 -19731.802,E2 -19731.802} C_VEL
LIN {X 0,Y 243.834,Z 452.214,A -85,B 0,C 180,E1 -19732.728,E2 -19732.728} C_VEL
LIN {X 0,Y 242.405,Z 464.365,A -85,B 0,C 180,E1 -19734.061,E2 -19734.061} C_VEL
LIN {X 0,Y 240.687,Z 476.602,A -85,B 0,C 180,E1 -19735.81,E2 -19735.81} C_VEL
LIN {X 0,Y 239.049,Z 487.356,A -85,B 0,C 180,E1 -19737.774,E2 -19737.774} C_VEL
LIN {X 0,Y 237.38,Z 496.992,A -85,B 0,C 180,E1 -19739.975,E2 -19739.975} C_VEL
LIN {X 0,Y 235.89,Z 505.637,A -85,B 0,C 180,E1 -19742.432,E2 -19742.432} C_VEL
LIN {X 0,Y 234.517,Z 513.512,A -85,B 0,C 180,E1 -19745.295,E2 -19745.295} C_VEL
LIN {X 0,Y 233.795,Z 518.78,A -85,B 0,C 180,E1 -19747.723,E2 -19747.723} C_VEL
LIN {X 0,Y 233.207,Z 522.911,A -85,B 0,C 180,E1 -19750.122,E2 -19750.122} C_VEL
LIN {X 0,Y 232.554,Z 527.161,A -85,B 0,C 180,E1 -19753.505,E2 -19753.505} C_VEL
LIN {X 0,Y 232.425,Z 529.479,A -85,B 0,C 180,E1 -19756.528,E2 -19756.528} C_VEL
LIN {X 0,Y 232.564,Z 530.476,A -85,B 0,C 180,E1 -19759.069,E2 -19759.069} C_VEL
LIN {X 0,Y 232.929,Z 530.577,A -85,B 0,C 180,E1 -19761.674,E2 -19761.674} C_VEL
LIN {X 0,Y 233.846,Z 529.244,A -85,B 0,C 180,E1 -19765.177,E2 -19765.177} C_VEL
LIN {X 0,Y 235.258,Z 526.464,A -85,B 0,C 180,E1 -19768.48,E2 -19768.48} C_VEL
LIN {X 0,Y 237.18,Z 522.092,A -85,B 0,C 180,E1 -19771.698,E2 -19771.698} C_VEL
LIN {X 0,Y 239.485,Z 516.619,A -85,B 0,C 180,E1 -19774.574,E2 -19774.574} C_VEL
LIN {X 0,Y 241.78,Z 510.871,A -85,B 0,C 180,E1 -19776.895,E2 -19776.895} C_VEL
LIN {X 0,Y 244.659,Z 503.069,A -85,B 0,C 180,E1 -19779.396,E2 -19779.396} C_VEL
LIN {X 0,Y 247.466,Z 494.778,A -85,B 0,C 180,E1 -19781.502,E2 -19781.502} C_VEL
LIN {X 0,Y 250.475,Z 484.962,A -85,B 0,C 180,E1 -19783.492,E2 -19783.492} C_VEL
LIN {X 0,Y 253.253,Z 474.805,A -85,B 0,C 180,E1 -19785.126,E2 -19785.126} C_VEL
LIN {X 0,Y 256.085,Z 462.818,A -85,B 0,C 180,E1 -19786.611,E2 -19786.611} C_VEL
LIN {X 0,Y 258.355,Z 450.27,A -85,B 0,C 180,E1 -19787.817,E2 -19787.817} C_VEL
LIN {X 0,Y 259.922,Z 438.382,A -85,B 0,C 180,E1 -19788.662,E2 -19788.662} C_VEL
LIN {X 0,Y 261.24,Z 425.13,A -85,B 0,C 180,E1 -19789.277,E2 -19789.277} C_VEL
LIN {X 0,Y 264.907,Z 370.247,A -85,B 0,C 180,E1 -19791.056,E2 -19791.056} C_VEL
LIN {X 0,Y 260.153,Z 359.919,A -85,B 0,C 180,E1 -19792.603,E2 -19792.603} C_VEL
LIN {X 0,Y 254.092,Z 348.637,A -85,B 0,C 180,E1 -19794.712,E2 -19794.712} C_VEL
LIN {X 0,Y 249.96,Z 341.936,A -85,B 0,C 180,E1 -19796.241,E2 -19796.241} C_VEL
LIN {X 0,Y 242.379,Z 330.944,A -85,B 0,C 180,E1 -19799.377,E2 -19799.377} C_VEL
LIN {X 0,Y 240.251,Z 328.032,A -85,B 0,C 180,E1 -19800.367,E2 -19800.367} C_VEL
LIN {X 0,Y 238.343,Z 325.916,A -85,B 0,C 180,E1 -19801.267,E2 -19801.267} C_VEL
LIN {X 0,Y 236.113,Z 323.353,A -85,B 0,C 180,E1 -19802.399,E2 -19802.399} C_VEL
LIN {X 0,Y 235.647,Z 322.348,A -85,B 0,C 180,E1 -19802.778,E2 -19802.778} C_VEL
LIN {X 0,Y 235.263,Z 321.172,A -85,B 0,C 180,E1 -19803.854,E2 -19803.854} C_VEL
LIN {X 0,Y 235.363,Z 321.158,A -85,B 0,C 180,E1 -19806.859,E2 -19806.859} C_VEL
LIN {X 0,Y 235.303,Z 321.171,A -85,B 0,C 180,E1 -19808.955,E2 -19808.955} C_VEL
LIN {X 0,Y 234.583,Z 321.256,A -85,B 0,C 180,E1 -19810.382,E2 -19810.382} C_VEL
LIN {X 0,Y 231.657,Z 321.622,A -85,B 0,C 180,E1 -19812.706,E2 -19812.706} C_VEL
LIN {X 0,Y 229.18,Z 321.934,A -85,B 0,C 180,E1 -19814.601,E2 -19814.601} C_VEL
LIN {X 0,Y 228.101,Z 322.068,A -85,B 0,C 180,E1 -19816.074,E2 -19816.074} C_VEL
LIN {X 0,Y 228.002,Z 322.075,A -85,B 0,C 180,E1 -19816.574,E2 -19816.574} C_VEL
LIN {X 0,Y 227.947,Z 322.082,A -85,B 0,C 180,E1 -19821.714,E2 -19821.714} C_VEL
LIN {X 0,Y 227.945,Z 322.088,A -85,B 0,C 180,E1 -19826.602,E2 -19826.602} C_VEL
LIN {X 0,Y 227.91,Z 322.091,A -85,B 0,C 180,E1 -19830.295,E2 -19830.295} C_VEL
LIN {X 0,Y 227.898,Z 322.168,A -85,B 0,C 180,E1 -19834.517,E2 -19834.517} C_VEL
LIN {X 0,Y 229.077,Z 325.158,A -85,B 0,C 180,E1 -19837.85,E2 -19837.85} C_VEL
LIN {X 0,Y 230.715,Z 330.063,A -85,B 0,C 180,E1 -19842.079,E2 -19842.079} C_VEL
LIN {X 0,Y 234.996,Z 336.176,A -85,B 0,C 180,E1 -19844.557,E2 -19844.557} C_VEL
LIN {X 0,Y 239.999,Z 343.745,A -85,B 0,C 180,E1 -19847.061,E2 -19847.061} C_VEL
LIN {X 0,Y 243.731,Z 349.894,A -85,B 0,C 180,E1 -19848.746,E2 -19848.746} C_VEL
LIN {X 0,Y 248.293,Z 357.926,A -85,B 0,C 180,E1 -19850.63,E2 -19850.63} C_VEL
LIN {X 0,Y 253.824,Z 369.422,A -85,B 0,C 180,E1 -19852.757,E2 -19852.757} C_VEL
LIN {X 0,Y 257.169,Z 377.775,A -85,B 0,C 180,E1 -19854.016,E2 -19854.016} C_VEL
LIN {X 0,Y 258.64,Z 391.733,A -85,B 0,C 180,E1 -19855.027,E2 -19855.027} C_VEL
LIN {X 0,Y 255.511,Z 438.357,A -85,B 0,C 180,E1 -19856.584,E2 -19856.584} C_VEL
LIN {X 0,Y 253.952,Z 452.343,A -85,B 0,C 180,E1 -19857.221,E2 -19857.221} C_VEL
LIN {X 0,Y 251.569,Z 466.083,A -85,B 0,C 180,E1 -19858.176,E2 -19858.176} C_VEL
LIN {X 0,Y 249.121,Z 477.307,A -85,B 0,C 180,E1 -19859.247,E2 -19859.247} C_VEL
LIN {X 0,Y 246.044,Z 489.13,A -85,B 0,C 180,E1 -19860.714,E2 -19860.714} C_VEL
LIN {X 0,Y 243.518,Z 497.62,A -85,B 0,C 180,E1 -19862.031,E2 -19862.031} C_VEL
LIN {X 0,Y 240.196,Z 507.646,A -85,B 0,C 180,E1 -19863.966,E2 -19863.966} C_VEL
LIN {X 0,Y 236.793,Z 517.397,A -85,B 0,C 180,E1 -19866.378,E2 -19866.378} C_VEL
LIN {X 0,Y 233.742,Z 525.29,A -85,B 0,C 180,E1 -19868.849,E2 -19868.849} C_VEL
LIN {X 0,Y 231.395,Z 531.641,A -85,B 0,C 180,E1 -19871.402,E2 -19871.402} C_VEL
LIN {X 0,Y 229.24,Z 536.78,A -85,B 0,C 180,E1 -19873.982,E2 -19873.982} C_VEL
LIN {X 0,Y 227.622,Z 540.799,A -85,B 0,C 180,E1 -19876.61,E2 -19876.61} C_VEL
LIN {X 0,Y 226.592,Z 543.8,A -85,B 0,C 180,E1 -19879.274,E2 -19879.274} C_VEL
LIN {X 0,Y 225.808,Z 546.305,A -85,B 0,C 180,E1 -19882.847,E2 -19882.847} C_VEL
LIN {X 0,Y 225.638,Z 547.108,A -85,B 0,C 180,E1 -19885.352,E2 -19885.352} C_VEL
LIN {X 0,Y 225.722,Z 547.055,A -85,B 0,C 180,E1 -19888.215,E2 -19888.215} C_VEL
LIN {X 0,Y 225.819,Z 546.48,A -85,B 0,C 180,E1 -19889.999,E2 -19889.999} C_VEL
LIN {X 0,Y 225.785,Z 545.49,A -85,B 0,C 180,E1 -19891.783,E2 -19891.783} C_VEL
LIN {X 0,Y 225.758,Z 542.538,A -85,B 0,C 180,E1 -19895.009,E2 -19895.009} C_VEL
LIN {X 0,Y 225.992,Z 538.348,A -85,B 0,C 180,E1 -19898.043,E2 -19898.043} C_VEL
LIN {X 0,Y 226.483,Z 533.389,A -85,B 0,C 180,E1 -19900.729,E2 -19900.729} C_VEL
LIN {X 0,Y 227.331,Z 527.095,A -85,B 0,C 180,E1 -19903.406,E2 -19903.406} C_VEL
LIN {X 0,Y 228.633,Z 519.212,A -85,B 0,C 180,E1 -19906.059,E2 -19906.059} C_VEL
LIN {X 0,Y 229.971,Z 511.681,A -85,B 0,C 180,E1 -19908.112,E2 -19908.112} C_VEL
LIN {X 0,Y 231.772,Z 501.242,A -85,B 0,C 180,E1 -19910.407,E2 -19910.407} C_VEL
LIN {X 0,Y 233.323,Z 491.579,A -85,B 0,C 180,E1 -19912.117,E2 -19912.117} C_VEL
LIN {X 0,Y 234.94,Z 481.272,A -85,B 0,C 180,E1 -19913.583,E2 -19913.583} C_VEL
LIN {X 0,Y 236.579,Z 469.085,A -85,B 0,C 180,E1 -19914.926,E2 -19914.926} C_VEL
LIN {X 0,Y 238.04,Z 455.859,A -85,B 0,C 180,E1 -19915.991,E2 -19915.991} C_VEL
LIN {X 0,Y 239.008,Z 442.81,A -85,B 0,C 180,E1 -19916.7,E2 -19916.7} C_VEL
LIN {X 0,Y 241.222,Z 386.695,A -85,B 0,C 180,E1 -19918.631,E2 -19918.631} C_VEL
LIN {X 0,Y 236.918,Z 353.232,A -85,B 0,C 180,E1 -19920.316,E2 -19920.316} C_VEL
LIN {X 0,Y 230.767,Z 335.634,A -85,B 0,C 180,E1 -19921.673,E2 -19921.673} C_VEL
LIN {X 0,Y 228.764,Z 325.813,A -85,B 0,C 180,E1 -19925.71,E2 -19925.71} C_VEL
LIN {X 0,Y 227.941,Z 322.097,A -85,B 0,C 180,E1 -19927.326,E2 -19927.326} C_VEL
LIN {X 0,Y 227.804,Z 322.11,A -85,B 0,C 180,E1 -19932.233,E2 -19932.233} C_VEL
LIN {X 0,Y 227.822,Z 322.105,A -85,B 0,C 180,E1 -19935.194,E2 -19935.194} C_VEL
LIN {X 0,Y 227.828,Z 322.105,A -85,B 0,C 180,E1 -19939.624,E2 -19939.624} C_VEL
LIN {X 0,Y 227.896,Z 322.096,A -85,B 0,C 180,E1 -19944.131,E2 -19944.131} C_VEL
LIN {X 0,Y 227.868,Z 322.091,A -85,B 0,C 180,E1 -19948.378,E2 -19948.378} C_VEL
LIN {X 0,Y 227.881,Z 322.093,A -85,B 0,C 180,E1 -19952.445,E2 -19952.445} C_VEL
LIN {X 0,Y 227.91,Z 322.096,A -85,B 0,C 180,E1 -19956.367,E2 -19956.367} C_VEL
LIN {X 0,Y 227.938,Z 322.086,A -85,B 0,C 180,E1 -19960.174,E2 -19960.174} C_VEL
LIN {X 0,Y 228.053,Z 322.077,A -85,B 0,C 180,E1 -19963.898,E2 -19963.898} C_VEL
LIN {X 0,Y 228.089,Z 322.066,A -85,B 0,C 180,E1 -19967.544,E2 -19967.544} C_VEL
LIN {X 0,Y 228.301,Z 322.044,A -85,B 0,C 180,E1 -19971.146,E2 -19971.146} C_VEL
LIN {X 0,Y 228.35,Z 322.039,A -85,B 0,C 180,E1 -19972.929,E2 -19972.929} C_VEL
LIN {X 0,Y 228.549,Z 322.004,A -85,B 0,C 180,E1 -19978.238,E2 -19978.238} C_VEL
LIN {X 0,Y 228.548,Z 322.011,A -85,B 0,C 180,E1 -19981.763,E2 -19981.763} C_VEL
LIN {X 0,Y 228.307,Z 322.041,A -85,B 0,C 180,E1 -19987.073,E2 -19987.073} C_VEL
LIN {X 0,Y 228.141,Z 322.052,A -85,B 0,C 180,E1 -19990.652,E2 -19990.652} C_VEL
LIN {X 0,Y 228.061,Z 322.07,A -85,B 0,C 180,E1 -19994.273,E2 -19994.273} C_VEL
LIN {X 0,Y 227.999,Z 322.082,A -85,B 0,C 180,E1 -19997.954,E2 -19997.954} C_VEL
LIN {X 0,Y 227.917,Z 322.088,A -85,B 0,C 180,E1 -20002.325,E2 -20002.325} C_VEL
LIN {X 0,Y 227.919,Z 322.082,A -85,B 0,C 180,E1 -20006.593,E2 -20006.593} C_VEL
LIN {X 0,Y 227.87,Z 322.097,A -85,B 0,C 180,E1 -20010.282,E2 -20010.282} C_VEL
LIN {X 0,Y 227.874,Z 322.098,A -85,B 0,C 180,E1 -20013.722,E2 -20013.722} C_VEL
LIN {X 0,Y 227.841,Z 322.096,A -85,B 0,C 180,E1 -20018.092,E2 -20018.092} C_VEL
LIN {X 0,Y 227.804,Z 322.103,A -85,B 0,C 180,E1 -20022.745,E2 -20022.745} C_VEL
LIN {X 0,Y 227.798,Z 322.109,A -85,B 0,C 180,E1 -20027.256,E2 -20027.256} C_VEL
LIN {X 0,Y 227.843,Z 322.092,A -85,B 0,C 180,E1 -20031.91,E2 -20031.91} C_VEL
LIN {X 0,Y 227.879,Z 322.096,A -85,B 0,C 180,E1 -20036.379,E2 -20036.379} C_VEL
LIN {X 0,Y 227.877,Z 322.096,A -85,B 0,C 180,E1 -20040.433,E2 -20040.433} C_VEL
LIN {X 0,Y 227.903,Z 322.094,A -85,B 0,C 180,E1 -20044.424,E2 -20044.424} C_VEL
LIN {X 0,Y 227.953,Z 322.088,A -85,B 0,C 180,E1 -20048.287,E2 -20048.287} C_VEL
LIN {X 0,Y 228.026,Z 322.081,A -85,B 0,C 180,E1 -20053.897,E2 -20053.897} C_VEL
LIN {X 0,Y 228.069,Z 322.075,A -85,B 0,C 180,E1 -20057.544,E2 -20057.544} C_VEL
LIN {X 0,Y 228.26,Z 322.048,A -85,B 0,C 180,E1 -20061.145,E2 -20061.145} C_VEL
LIN {X 0,Y 228.308,Z 322.044,A -85,B 0,C 180,E1 -20062.928,E2 -20062.928} C_VEL
LIN {X 0,Y 228.502,Z 322.025,A -85,B 0,C 180,E1 -20068.239,E2 -20068.239} C_VEL
LIN {X 0,Y 228.501,Z 322.023,A -85,B 0,C 180,E1 -20071.764,E2 -20071.764} C_VEL
LIN {X 0,Y 228.297,Z 322.047,A -85,B 0,C 180,E1 -20077.074,E2 -20077.074} C_VEL
LIN {X 0,Y 228.127,Z 322.07,A -85,B 0,C 180,E1 -20080.653,E2 -20080.653} C_VEL
LIN {X 0,Y 227.998,Z 322.087,A -85,B 0,C 180,E1 -20085.19,E2 -20085.19} C_VEL
LIN {X 0,Y 229.147,Z 325.168,A -85,B 0,C 180,E1 -20085.482,E2 -20085.482} C_VEL
LIN {X 0,Y 235.235,Z 339.73,A -85,B 0,C 180,E1 -20086.713,E2 -20086.713} C_VEL
LIN {X 0,Y 242.068,Z 359.17,A -85,B 0,C 180,E1 -20088.134,E2 -20088.134} C_VEL
LIN {X 0,Y 239.148,Z 427.76,A -85,B 0,C 180,E1 -20090.494,E2 -20090.494} C_VEL
LIN {X 0,Y 238.072,Z 441.593,A -85,B 0,C 180,E1 -20091.314,E2 -20091.314} C_VEL
LIN {X 0,Y 236.941,Z 453.432,A -85,B 0,C 180,E1 -20092.337,E2 -20092.337} C_VEL
LIN {X 0,Y 235.364,Z 466.108,A -85,B 0,C 180,E1 -20093.809,E2 -20093.809} C_VEL
LIN {X 0,Y 233.664,Z 477.629,A -85,B 0,C 180,E1 -20095.533,E2 -20095.533} C_VEL
LIN {X 0,Y 231.946,Z 488.511,A -85,B 0,C 180,E1 -20097.621,E2 -20097.621} C_VEL
LIN {X 0,Y 230.183,Z 498.431,A -85,B 0,C 180,E1 -20099.999,E2 -20099.999} C_VEL
LIN {X 0,Y 228.713,Z 506.805,A -85,B 0,C 180,E1 -20102.531,E2 -20102.531} C_VEL
LIN {X 0,Y 227.355,Z 514.373,A -85,B 0,C 180,E1 -20105.423,E2 -20105.423} C_VEL
LIN {X 0,Y 226.532,Z 520.314,A -85,B 0,C 180,E1 -20108.353,E2 -20108.353} C_VEL
LIN {X 0,Y 225.912,Z 524.127,A -85,B 0,C 180,E1 -20110.792,E2 -20110.792} C_VEL
LIN {X 0,Y 225.388,Z 527.913,A -85,B 0,C 180,E1 -20114.177,E2 -20114.177} C_VEL
LIN {X 0,Y 225.327,Z 529.715,A -85,B 0,C 180,E1 -20116.67,E2 -20116.67} C_VEL
LIN {X 0,Y 225.471,Z 530.688,A -85,B 0,C 180,E1 -20119.112,E2 -20119.112} C_VEL
LIN {X 0,Y 225.798,Z 530.891,A -85,B 0,C 180,E1 -20121.5,E2 -20121.5} C_VEL
LIN {X 0,Y 226.339,Z 530.421,A -85,B 0,C 180,E1 -20123.845,E2 -20123.845} C_VEL
LIN {X 0,Y 227.273,Z 528.949,A -85,B 0,C 180,E1 -20126.609,E2 -20126.609} C_VEL
LIN {X 0,Y 228.61,Z 526.405,A -85,B 0,C 180,E1 -20129.406,E2 -20129.406} C_VEL
LIN {X 0,Y 230.393,Z 522.683,A -85,B 0,C 180,E1 -20132.207,E2 -20132.207} C_VEL
LIN {X 0,Y 232.671,Z 517.68,A -85,B 0,C 180,E1 -20134.983,E2 -20134.983} C_VEL
LIN {X 0,Y 235.457,Z 511.227,A -85,B 0,C 180,E1 -20137.715,E2 -20137.715} C_VEL
LIN {X 0,Y 238.019,Z 504.724,A -85,B 0,C 180,E1 -20139.893,E2 -20139.893} C_VEL
LIN {X 0,Y 241.13,Z 496.204,A -85,B 0,C 180,E1 -20142.18,E2 -20142.18} C_VEL
LIN {X 0,Y 244.148,Z 487.028,A -85,B 0,C 180,E1 -20144.129,E2 -20144.129} C_VEL
LIN {X 0,Y 247.06,Z 477.117,A -85,B 0,C 180,E1 -20145.813,E2 -20145.813} C_VEL
LIN {X 0,Y 249.948,Z 465.855,A -85,B 0,C 180,E1 -20147.332,E2 -20147.332} C_VEL
LIN {X 0,Y 252.382,Z 454.117,A -85,B 0,C 180,E1 -20148.549,E2 -20148.549} C_VEL
LIN {X 0,Y 254.329,Z 441.475,A -85,B 0,C 180,E1 -20149.539,E2 -20149.539} C_VEL
LIN {X 0,Y 255.805,Z 429.148,A -85,B 0,C 180,E1 -20150.188,E2 -20150.188} C_VEL
LIN {X 0,Y 259.716,Z 372.727,A -85,B 0,C 180,E1 -20152.081,E2 -20152.081} C_VEL
LIN {X 0,Y 255.732,Z 363.967,A -85,B 0,C 180,E1 -20153.48,E2 -20153.48} C_VEL
LIN {X 0,Y 250.214,Z 353.498,A -85,B 0,C 180,E1 -20155.502,E2 -20155.502} C_VEL
LIN {X 0,Y 246.082,Z 346.749,A -85,B 0,C 180,E1 -20157.135,E2 -20157.135} C_VEL
LIN {X 0,Y 239.567,Z 336.945,A -85,B 0,C 180,E1 -20160,E2 -20160} C_VEL
LIN {X 0,Y 236.428,Z 332.671,A -85,B 0,C 180,E1 -20161.54,E2 -20161.54} C_VEL
LIN {X 0,Y 233.713,Z 329.699,A -85,B 0,C 180,E1 -20162.962,E2 -20162.962} C_VEL
LIN {X 0,Y 232.414,Z 327.942,A -85,B 0,C 180,E1 -20163.711,E2 -20163.711} C_VEL
LIN {X 0,Y 229.477,Z 325.311,A -85,B 0,C 180,E1 -20165.437,E2 -20165.437} C_VEL
LIN {X 0,Y 228.477,Z 323.131,A -85,B 0,C 180,E1 -20166.291,E2 -20166.291} C_VEL
LIN {X 0,Y 228.279,Z 322.041,A -85,B 0,C 180,E1 -20167.518,E2 -20167.518} C_VEL
LIN {X 0,Y 228.148,Z 322.057,A -85,B 0,C 180,E1 -20170.651,E2 -20170.651} C_VEL
LIN {X 0,Y 228.048,Z 322.069,A -85,B 0,C 180,E1 -20174.273,E2 -20174.273} C_VEL
LIN {X 0,Y 228.002,Z 322.075,A -85,B 0,C 180,E1 -20176.574,E2 -20176.574} C_VEL
LIN {X 0,Y 227.31,Z 322.164,A -85,B 0,C 180,E1 -20178.046,E2 -20178.046} C_VEL
LIN {X 0,Y 224.464,Z 322.514,A -85,B 0,C 180,E1 -20180.449,E2 -20180.449} C_VEL
LIN {X 0,Y 221.213,Z 322.923,A -85,B 0,C 180,E1 -20183.418,E2 -20183.418} C_VEL
LIN {X 0,Y 220.864,Z 322.961,A -85,B 0,C 180,E1 -20184.446,E2 -20184.446} C_VEL
LIN {X 0,Y 220.826,Z 322.967,A -85,B 0,C 180,E1 -20188.644,E2 -20188.644} C_VEL
LIN {X 0,Y 222.247,Z 326.64,A -85,B 0,C 180,E1 -20194.695,E2 -20194.695} C_VEL
LIN {X 0,Y 223.365,Z 329.335,A -85,B 0,C 180,E1 -20197.681,E2 -20197.681} C_VEL
LIN {X 0,Y 226.36,Z 333.98,A -85,B 0,C 180,E1 -20200.096,E2 -20200.096} C_VEL
LIN {X 0,Y 228.854,Z 337.088,A -85,B 0,C 180,E1 -20201.76,E2 -20201.76} C_VEL
LIN {X 0,Y 233.395,Z 343.757,A -85,B 0,C 180,E1 -20204.457,E2 -20204.457} C_VEL
LIN {X 0,Y 237.241,Z 349.887,A -85,B 0,C 180,E1 -20206.46,E2 -20206.46} C_VEL
LIN {X 0,Y 240.437,Z 355.319,A -85,B 0,C 180,E1 -20207.99,E2 -20207.99} C_VEL
LIN {X 0,Y 244.782,Z 363.264,A -85,B 0,C 180,E1 -20209.89,E2 -20209.89} C_VEL
LIN {X 0,Y 250.064,Z 374.706,A -85,B 0,C 180,E1 -20212.057,E2 -20212.057} C_VEL
LIN {X 0,Y 252.538,Z 381.217,A -85,B 0,C 180,E1 -20213.049,E2 -20213.049} C_VEL
LIN {X 0,Y 253.623,Z 393.142,A -85,B 0,C 180,E1 -20213.942,E2 -20213.942} C_VEL
LIN {X 0,Y 249.966,Z 443.052,A -85,B 0,C 180,E1 -20215.662,E2 -20215.662} C_VEL
LIN {X 0,Y 248.14,Z 456.098,A -85,B 0,C 180,E1 -20216.353,E2 -20216.353} C_VEL
LIN {X 0,Y 245.665,Z 468.794,A -85,B 0,C 180,E1 -20217.317,E2 -20217.317} C_VEL
LIN {X 0,Y 242.763,Z 480.89,A -85,B 0,C 180,E1 -20218.593,E2 -20218.593} C_VEL
LIN {X 0,Y 239.578,Z 491.896,A -85,B 0,C 180,E1 -20220.086,E2 -20220.086} C_VEL
LIN {X 0,Y 236.319,Z 501.951,A -85,B 0,C 180,E1 -20221.827,E2 -20221.827} C_VEL
LIN {X 0,Y 232.704,Z 511.91,A -85,B 0,C 180,E1 -20224.028,E2 -20224.028} C_VEL
LIN {X 0,Y 229.216,Z 520.8,A -85,B 0,C 180,E1 -20226.509,E2 -20226.509} C_VEL
LIN {X 0,Y 226.04,Z 528.533,A -85,B 0,C 180,E1 -20229.3,E2 -20229.3} C_VEL
LIN {X 0,Y 223.904,Z 533.775,A -85,B 0,C 180,E1 -20231.706,E2 -20231.706} C_VEL
LIN {X 0,Y 221.753,Z 538.389,A -85,B 0,C 180,E1 -20234.371,E2 -20234.371} C_VEL
LIN {X 0,Y 220.299,Z 541.94,A -85,B 0,C 180,E1 -20237.095,E2 -20237.095} C_VEL
LIN {X 0,Y 219.087,Z 545.145,A -85,B 0,C 180,E1 -20240.769,E2 -20240.769} C_VEL
LIN {X 0,Y 218.735,Z 546.154,A -85,B 0,C 180,E1 -20242.615,E2 -20242.615} C_VEL
LIN {X 0,Y 218.547,Z 546.897,A -85,B 0,C 180,E1 -20245.48,E2 -20245.48} C_VEL
LIN {X 0,Y 218.634,Z 546.712,A -85,B 0,C 180,E1 -20248.157,E2 -20248.157} C_VEL
LIN {X 0,Y 218.751,Z 546.095,A -85,B 0,C 180,E1 -20249.999,E2 -20249.999} C_VEL
LIN {X 0,Y 218.695,Z 545.047,A -85,B 0,C 180,E1 -20251.84,E2 -20251.84} C_VEL
LIN {X 0,Y 218.693,Z 542.199,A -85,B 0,C 180,E1 -20254.978,E2 -20254.978} C_VEL
LIN {X 0,Y 218.927,Z 537.679,A -85,B 0,C 180,E1 -20258.305,E2 -20258.305} C_VEL
LIN {X 0,Y 219.47,Z 532.61,A -85,B 0,C 180,E1 -20261.076,E2 -20261.076} C_VEL
LIN {X 0,Y 220.398,Z 526.191,A -85,B 0,C 180,E1 -20263.836,E2 -20263.836} C_VEL
LIN {X 0,Y 221.755,Z 518.099,A -85,B 0,C 180,E1 -20266.572,E2 -20266.572} C_VEL
LIN {X 0,Y 223.14,Z 510.137,A -85,B 0,C 180,E1 -20268.751,E2 -20268.751} C_VEL
LIN {X 0,Y 225.071,Z 499.758,A -85,B 0,C 180,E1 -20271.043,E2 -20271.043} C_VEL
LIN {X 0,Y 226.741,Z 489.825,A -85,B 0,C 180,E1 -20272.794,E2 -20272.794} C_VEL
LIN {X 0,Y 228.369,Z 479.078,A -85,B 0,C 180,E1 -20274.305,E2 -20274.305} C_VEL
LIN {X 0,Y 229.961,Z 467.432,A -85,B 0,C 180,E1 -20275.573,E2 -20275.573} C_VEL
LIN {X 0,Y 231.399,Z 454.49,A -85,B 0,C 180,E1 -20276.613,E2 -20276.613} C_VEL
LIN {X 0,Y 232.335,Z 441.905,A -85,B 0,C 180,E1 -20277.287,E2 -20277.287} C_VEL
LIN {X 0,Y 234.548,Z 387.085,A -85,B 0,C 180,E1 -20279.227,E2 -20279.227} C_VEL
LIN {X 0,Y 230.579,Z 355.596,A -85,B 0,C 180,E1 -20280.87,E2 -20280.87} C_VEL
LIN {X 0,Y 223.484,Z 335.362,A -85,B 0,C 180,E1 -20282.487,E2 -20282.487} C_VEL
LIN {X 0,Y 221.572,Z 325.997,A -85,B 0,C 180,E1 -20286.491,E2 -20286.491} C_VEL
LIN {X 0,Y 220.895,Z 322.974,A -85,B 0,C 180,E1 -20287.909,E2 -20287.909} C_VEL
LIN {X 0,Y 220.758,Z 322.987,A -85,B 0,C 180,E1 -20292.927,E2 -20292.927} C_VEL
LIN {X 0,Y 220.76,Z 322.987,A -85,B 0,C 180,E1 -20297.071,E2 -20297.071} C_VEL
LIN {X 0,Y 220.805,Z 322.982,A -85,B 0,C 180,E1 -20300.463,E2 -20300.463} C_VEL
LIN {X 0,Y 220.828,Z 322.978,A -85,B 0,C 180,E1 -20302.794,E2 -20302.794} C_VEL
LIN {X 0,Y 220.82,Z 322.971,A -85,B 0,C 180,E1 -20307.245,E2 -20307.245} C_VEL
LIN {X 0,Y 220.832,Z 322.971,A -85,B 0,C 180,E1 -20311.486,E2 -20311.486} C_VEL
LIN {X 0,Y 220.863,Z 322.974,A -85,B 0,C 180,E1 -20315.565,E2 -20315.565} C_VEL
LIN {X 0,Y 220.888,Z 322.966,A -85,B 0,C 180,E1 -20319.514,E2 -20319.514} C_VEL
LIN {X 0,Y 221.012,Z 322.957,A -85,B 0,C 180,E1 -20323.37,E2 -20323.37} C_VEL
LIN {X 0,Y 221.107,Z 322.934,A -85,B 0,C 180,E1 -20329.006,E2 -20329.006} C_VEL
LIN {X 0,Y 221.285,Z 322.918,A -85,B 0,C 180,E1 -20332.702,E2 -20332.702} C_VEL
LIN {X 0,Y 221.507,Z 322.881,A -85,B 0,C 180,E1 -20338.182,E2 -20338.182} C_VEL
LIN {X 0,Y 221.506,Z 322.889,A -85,B 0,C 180,E1 -20341.819,E2 -20341.819} C_VEL
LIN {X 0,Y 221.243,Z 322.921,A -85,B 0,C 180,E1 -20347.3,E2 -20347.3} C_VEL
LIN {X 0,Y 221.063,Z 322.932,A -85,B 0,C 180,E1 -20350.997,E2 -20350.997} C_VEL
LIN {X 0,Y 220.992,Z 322.95,A -85,B 0,C 180,E1 -20354.74,E2 -20354.74} C_VEL
LIN {X 0,Y 220.916,Z 322.964,A -85,B 0,C 180,E1 -20358.55,E2 -20358.55} C_VEL
LIN {X 0,Y 220.864,Z 322.963,A -85,B 0,C 180,E1 -20362.666,E2 -20362.666} C_VEL
LIN {X 0,Y 220.862,Z 322.963,A -85,B 0,C 180,E1 -20367.006,E2 -20367.006} C_VEL
LIN {X 0,Y 220.815,Z 322.979,A -85,B 0,C 180,E1 -20370.76,E2 -20370.76} C_VEL
LIN {X 0,Y 220.798,Z 322.979,A -85,B 0,C 180,E1 -20374.956,E2 -20374.956} C_VEL
LIN {X 0,Y 220.804,Z 322.964,A -85,B 0,C 180,E1 -20379.538,E2 -20379.538} C_VEL
LIN {X 0,Y 220.765,Z 322.982,A -85,B 0,C 180,E1 -20384.457,E2 -20384.457} C_VEL
LIN {X 0,Y 220.757,Z 322.984,A -85,B 0,C 180,E1 -20388.046,E2 -20388.046} C_VEL
LIN {X 0,Y 220.824,Z 322.967,A -85,B 0,C 180,E1 -20392.794,E2 -20392.794} C_VEL
LIN {X 0,Y 220.812,Z 322.98,A -85,B 0,C 180,E1 -20397.245,E2 -20397.245} C_VEL
LIN {X 0,Y 220.805,Z 322.981,A -85,B 0,C 180,E1 -20401.483,E2 -20401.483} C_VEL
LIN {X 0,Y 220.848,Z 322.975,A -85,B 0,C 180,E1 -20405.564,E2 -20405.564} C_VEL
LIN {X 0,Y 220.88,Z 322.971,A -85,B 0,C 180,E1 -20409.514,E2 -20409.514} C_VEL
LIN {X 0,Y 220.982,Z 322.957,A -85,B 0,C 180,E1 -20413.369,E2 -20413.369} C_VEL
LIN {X 0,Y 221.006,Z 322.953,A -85,B 0,C 180,E1 -20417.139,E2 -20417.139} C_VEL
LIN {X 0,Y 221.2,Z 322.928,A -85,B 0,C 180,E1 -20420.86,E2 -20420.86} C_VEL
LIN {X 0,Y 221.246,Z 322.924,A -85,B 0,C 180,E1 -20422.701,E2 -20422.701} C_VEL
LIN {X 0,Y 221.439,Z 322.905,A -85,B 0,C 180,E1 -20428.182,E2 -20428.182} C_VEL
LIN {X 0,Y 221.545,Z 322.89,A -85,B 0,C 180,E1 -20430.001,E2 -20430.001} C_VEL
LIN {X 0,Y 221.438,Z 322.904,A -85,B 0,C 180,E1 -20431.82,E2 -20431.82} C_VEL
LIN {X 0,Y 221.234,Z 322.927,A -85,B 0,C 180,E1 -20437.301,E2 -20437.301} C_VEL
LIN {X 0,Y 221.05,Z 322.949,A -85,B 0,C 180,E1 -20440.998,E2 -20440.998} C_VEL
LIN {X 0,Y 220.953,Z 322.963,A -85,B 0,C 180,E1 -20444.448,E2 -20444.448} C_VEL
LIN {X 0,Y 221.984,Z 325.844,A -85,B 0,C 180,E1 -20444.702,E2 -20444.702} C_VEL
LIN {X 0,Y 228.755,Z 341.607,A -85,B 0,C 180,E1 -20446.105,E2 -20446.105} C_VEL
LIN {X 0,Y 235.46,Z 360.682,A -85,B 0,C 180,E1 -20447.553,E2 -20447.553} C_VEL
LIN {X 0,Y 232.459,Z 427.924,A -85,B 0,C 180,E1 -20449.93,E2 -20449.93} C_VEL
LIN {X 0,Y 231.395,Z 441.197,A -85,B 0,C 180,E1 -20450.729,E2 -20450.729} C_VEL
LIN {X 0,Y 230.15,Z 453.894,A -85,B 0,C 180,E1 -20451.849,E2 -20451.849} C_VEL
LIN {X 0,Y 228.482,Z 466.711,A -85,B 0,C 180,E1 -20453.385,E2 -20453.385} C_VEL
LIN {X 0,Y 226.697,Z 478.446,A -85,B 0,C 180,E1 -20455.21,E2 -20455.21} C_VEL
LIN {X 0,Y 224.86,Z 489.643,A -85,B 0,C 180,E1 -20457.453,E2 -20457.453} C_VEL
LIN {X 0,Y 223.115,Z 499.163,A -85,B 0,C 180,E1 -20459.838,E2 -20459.838} C_VEL
LIN {X 0,Y 221.494,Z 507.979,A -85,B 0,C 180,E1 -20462.644,E2 -20462.644} C_VEL
LIN {X 0,Y 220.221,Z 515.088,A -85,B 0,C 180,E1 -20465.503,E2 -20465.503} C_VEL
LIN {X 0,Y 219.395,Z 520.918,A -85,B 0,C 180,E1 -20468.541,E2 -20468.541} C_VEL
LIN {X 0,Y 218.731,Z 524.721,A -85,B 0,C 180,E1 -20471.101,E2 -20471.101} C_VEL
LIN {X 0,Y 218.343,Z 527.618,A -85,B 0,C 180,E1 -20473.702,E2 -20473.702} C_VEL
LIN {X 0,Y 218.239,Z 528.816,A -85,B 0,C 180,E1 -20475.112,E2 -20475.112} C_VEL
LIN {X 0,Y 218.272,Z 530.395,A -85,B 0,C 180,E1 -20477.781,E2 -20477.781} C_VEL
LIN {X 0,Y 218.546,Z 531.136,A -85,B 0,C 180,E1 -20480.516,E2 -20480.516} C_VEL
LIN {X 0,Y 219.089,Z 530.981,A -85,B 0,C 180,E1 -20483.319,E2 -20483.319} C_VEL
LIN {X 0,Y 219.98,Z 529.861,A -85,B 0,C 180,E1 -20486.168,E2 -20486.168} C_VEL
LIN {X 0,Y 221.547,Z 527.282,A -85,B 0,C 180,E1 -20489.498,E2 -20489.498} C_VEL
LIN {X 0,Y 223.805,Z 522.974,A -85,B 0,C 180,E1 -20492.969,E2 -20492.969} C_VEL
LIN {X 0,Y 226.661,Z 517.136,A -85,B 0,C 180,E1 -20496.228,E2 -20496.228} C_VEL
LIN {X 0,Y 229.589,Z 510.712,A -85,B 0,C 180,E1 -20498.919,E2 -20498.919} C_VEL
LIN {X 0,Y 232.86,Z 502.683,A -85,B 0,C 180,E1 -20501.524,E2 -20501.524} C_VEL
LIN {X 0,Y 236.249,Z 493.664,A -85,B 0,C 180,E1 -20503.838,E2 -20503.838} C_VEL
LIN {X 0,Y 239.744,Z 483.397,A -85,B 0,C 180,E1 -20505.887,E2 -20505.887} C_VEL
LIN {X 0,Y 243.1,Z 471.813,A -85,B 0,C 180,E1 -20507.689,E2 -20507.689} C_VEL
LIN {X 0,Y 245.955,Z 460.101,A -85,B 0,C 180,E1 -20509.087,E2 -20509.087} C_VEL
LIN {X 0,Y 248.43,Z 446.565,A -85,B 0,C 180,E1 -20510.306,E2 -20510.306} C_VEL
LIN {X 0,Y 250.093,Z 434.764,A -85,B 0,C 180,E1 -20511.052,E2 -20511.052} C_VEL
LIN {X 0,Y 251.423,Z 420.296,A -85,B 0,C 180,E1 -20511.63,E2 -20511.63} C_VEL
LIN {X 0,Y 254.688,Z 375.268,A -85,B 0,C 180,E1 -20513.151,E2 -20513.151} C_VEL
LIN {X 0,Y 250.427,Z 365.966,A -85,B 0,C 180,E1 -20514.754,E2 -20514.754} C_VEL
LIN {X 0,Y 245.107,Z 355.992,A -85,B 0,C 180,E1 -20516.881,E2 -20516.881} C_VEL
LIN {X 0,Y 240.753,Z 349.028,A -85,B 0,C 180,E1 -20518.745,E2 -20518.745} C_VEL
LIN {X 0,Y 236.701,Z 342.866,A -85,B 0,C 180,E1 -20520.678,E2 -20520.678} C_VEL
LIN {X 0,Y 234.057,Z 339.052,A -85,B 0,C 180,E1 -20522.056,E2 -20522.056} C_VEL
LIN {X 0,Y 231.16,Z 335.71,A -85,B 0,C 180,E1 -20523.649,E2 -20523.649} C_VEL
LIN {X 0,Y 229.931,Z 334.095,A -85,B 0,C 180,E1 -20524.382,E2 -20524.382} C_VEL
LIN {X 0,Y 227.429,Z 331.868,A -85,B 0,C 180,E1 -20525.93,E2 -20525.93} C_VEL
LIN {X 0,Y 225.834,Z 329.066,A -85,B 0,C 180,E1 -20527.15,E2 -20527.15} C_VEL
LIN {X 0,Y 222.279,Z 325.953,A -85,B 0,C 180,E1 -20529.963,E2 -20529.963} C_VEL
LIN {X 0,Y 221.368,Z 324.181,A -85,B 0,C 180,E1 -20530.981,E2 -20530.981} C_VEL
LIN {X 0,Y 220.986,Z 322.948,A -85,B 0,C 180,E1 -20533.33,E2 -20533.33} C_VEL
LIN {X 0,Y 220.932,Z 322.954,A -85,B 0,C 180,E1 -20537.383,E2 -20537.383} C_VEL
LIN {X 0,Y 220.867,Z 322.97,A -85,B 0,C 180,E1 -20542.447,E2 -20542.447} C_VEL
LIN {X 0,Y 220.864,Z 322.961,A -85,B 0,C 180,E1 -20544.446,E2 -20544.446} C_VEL
LIN {X 0,Y 220.297,Z 323.481,A -85,B 0,C 180,E1 -20545.966,E2 -20545.966} C_VEL
LIN {X 0,Y 218.243,Z 325.918,A -85,B 0,C 180,E1 -20548.423,E2 -20548.423} C_VEL
LIN {X 0,Y 216.901,Z 328.475,A -85,B 0,C 180,E1 -20550.391,E2 -20550.391} C_VEL
LIN {X 0,Y 216.853,Z 330.282,A -85,B 0,C 180,E1 -20551.892,E2 -20551.892} C_VEL
LIN {X 0,Y 217.124,Z 330.799,A -85,B 0,C 180,E1 -20552.394,E2 -20552.394} C_VEL
LIN {X 0,Y 220.4,Z 334.795,A -85,B 0,C 180,E1 -20556.151,E2 -20556.151} C_VEL
LIN {X 0,Y 221.67,Z 336.269,A -85,B 0,C 180,E1 -20557.319,E2 -20557.319} C_VEL
LIN {X 0,Y 224.734,Z 340.91,A -85,B 0,C 180,E1 -20559.841,E2 -20559.841} C_VEL
LIN {X 0,Y 226.75,Z 343.614,A -85,B 0,C 180,E1 -20561.251,E2 -20561.251} C_VEL
LIN {X 0,Y 230.836,Z 349.872,A -85,B 0,C 180,E1 -20563.806,E2 -20563.806} C_VEL
LIN {X 0,Y 234.385,Z 355.833,A -85,B 0,C 180,E1 -20565.782,E2 -20565.782} C_VEL
LIN {X 0,Y 237.416,Z 361.09,A -85,B 0,C 180,E1 -20567.302,E2 -20567.302} C_VEL
LIN {X 0,Y 241.445,Z 368.861,A -85,B 0,C 180,E1 -20569.184,E2 -20569.184} C_VEL
LIN {X 0,Y 246.097,Z 379.436,A -85,B 0,C 180,E1 -20571.235,E2 -20571.235} C_VEL
LIN {X 0,Y 247.992,Z 384.788,A -85,B 0,C 180,E1 -20572.051,E2 -20572.051} C_VEL
LIN {X 0,Y 248.793,Z 394.416,A -85,B 0,C 180,E1 -20572.786,E2 -20572.786} C_VEL
LIN {X 0,Y 245.01,Z 442.724,A -85,B 0,C 180,E1 -20574.478,E2 -20574.478} C_VEL
LIN {X 0,Y 243.082,Z 455.802,A -85,B 0,C 180,E1 -20575.178,E2 -20575.178} C_VEL
LIN {X 0,Y 240.752,Z 467.407,A -85,B 0,C 180,E1 -20576.061,E2 -20576.061} C_VEL
LIN {X 0,Y 237.661,Z 479.745,A -85,B 0,C 180,E1 -20577.337,E2 -20577.337} C_VEL
LIN {X 0,Y 234.358,Z 490.895,A -85,B 0,C 180,E1 -20578.848,E2 -20578.848} C_VEL
LIN {X 0,Y 231.611,Z 498.981,A -85,B 0,C 180,E1 -20580.205,E2 -20580.205} C_VEL
LIN {X 0,Y 227.663,Z 509.519,A -85,B 0,C 180,E1 -20582.415,E2 -20582.415} C_VEL
LIN {X 0,Y 223.95,Z 518.725,A -85,B 0,C 180,E1 -20584.933,E2 -20584.933} C_VEL
LIN {X 0,Y 220.609,Z 526.203,A -85,B 0,C 180,E1 -20587.524,E2 -20587.524} C_VEL
LIN {X 0,Y 217.992,Z 532.283,A -85,B 0,C 180,E1 -20590.212,E2 -20590.212} C_VEL
LIN {X 0,Y 215.606,Z 537.155,A -85,B 0,C 180,E1 -20592.939,E2 -20592.939} C_VEL
LIN {X 0,Y 213.761,Z 540.926,A -85,B 0,C 180,E1 -20595.724,E2 -20595.724} C_VEL
LIN {X 0,Y 212.612,Z 543.703,A -85,B 0,C 180,E1 -20598.559,E2 -20598.559} C_VEL
LIN {X 0,Y 211.669,Z 545.994,A -85,B 0,C 180,E1 -20602.367,E2 -20602.367} C_VEL
LIN {X 0,Y 211.473,Z 546.661,A -85,B 0,C 180,E1 -20605.565,E2 -20605.565} C_VEL
LIN {X 0,Y 211.547,Z 546.367,A -85,B 0,C 180,E1 -20608.095,E2 -20608.095} C_VEL
LIN {X 0,Y 211.685,Z 545.699,A -85,B 0,C 180,E1 -20609.999,E2 -20609.999} C_VEL
LIN {X 0,Y 211.608,Z 544.554,A -85,B 0,C 180,E1 -20611.902,E2 -20611.902} C_VEL
LIN {X 0,Y 211.6,Z 541.918,A -85,B 0,C 180,E1 -20614.859,E2 -20614.859} C_VEL
LIN {X 0,Y 211.784,Z 538.422,A -85,B 0,C 180,E1 -20617.627,E2 -20617.627} C_VEL
LIN {X 0,Y 212.24,Z 533.636,A -85,B 0,C 180,E1 -20620.492,E2 -20620.492} C_VEL
LIN {X 0,Y 213.032,Z 527.523,A -85,B 0,C 180,E1 -20623.351,E2 -20623.351} C_VEL
LIN {X 0,Y 214.426,Z 519.901,A -85,B 0,C 180,E1 -20626.175,E2 -20626.175} C_VEL
LIN {X 0,Y 215.887,Z 512.096,A -85,B 0,C 180,E1 -20628.505,E2 -20628.505} C_VEL
LIN {X 0,Y 217.598,Z 502.549,A -85,B 0,C 180,E1 -20630.809,E2 -20630.809} C_VEL
LIN {X 0,Y 219.458,Z 491.967,A -85,B 0,C 180,E1 -20632.847,E2 -20632.847} C_VEL
LIN {X 0,Y 221.105,Z 481.851,A -85,B 0,C 180,E1 -20634.406,E2 -20634.406} C_VEL
LIN {X 0,Y 222.899,Z 470.141,A -85,B 0,C 180,E1 -20635.816,E2 -20635.816} C_VEL
LIN {X 0,Y 224.308,Z 458.176,A -85,B 0,C 180,E1 -20636.894,E2 -20636.894} C_VEL
LIN {X 0,Y 225.521,Z 444.56,A -85,B 0,C 180,E1 -20637.741,E2 -20637.741} C_VEL
LIN {X 0,Y 227.96,Z 388.208,A -85,B 0,C 180,E1 -20639.827,E2 -20639.827} C_VEL
LIN {X 0,Y 224.043,Z 357.174,A -85,B 0,C 180,E1 -20641.492,E2 -20641.492} C_VEL
LIN {X 0,Y 216.205,Z 335.072,A -85,B 0,C 180,E1 -20643.363,E2 -20643.363} C_VEL
LIN {X 0,Y 214.31,Z 326.141,A -85,B 0,C 180,E1 -20647.332,E2 -20647.332} C_VEL
LIN {X 0,Y 213.831,Z 323.854,A -85,B 0,C 180,E1 -20648.422,E2 -20648.422} C_VEL
LIN {X 0,Y 213.699,Z 323.865,A -85,B 0,C 180,E1 -20653.678,E2 -20653.678} C_VEL
LIN {X 0,Y 213.699,Z 323.864,A -85,B 0,C 180,E1 -20656.344,E2 -20656.344} C_VEL
LIN {X 0,Y 213.732,Z 323.861,A -85,B 0,C 180,E1 -20661.335,E2 -20661.335} C_VEL
LIN {X 0,Y 213.765,Z 323.855,A -85,B 0,C 180,E1 -20666.02,E2 -20666.02} C_VEL
LIN {X 0,Y 213.776,Z 323.837,A -85,B 0,C 180,E1 -20670.454,E2 -20670.454} C_VEL
LIN {X 0,Y 213.797,Z 323.854,A -85,B 0,C 180,E1 -20674.701,E2 -20674.701} C_VEL
LIN {X 0,Y 213.808,Z 323.85,A -85,B 0,C 180,E1 -20678.803,E2 -20678.803} C_VEL
LIN {X 0,Y 213.939,Z 323.835,A -85,B 0,C 180,E1 -20682.804,E2 -20682.804} C_VEL
LIN {X 0,Y 213.976,Z 323.827,A -85,B 0,C 180,E1 -20686.708,E2 -20686.708} C_VEL
LIN {X 0,Y 214.163,Z 323.803,A -85,B 0,C 180,E1 -20690.557,E2 -20690.557} C_VEL
LIN {X 0,Y 214.223,Z 323.798,A -85,B 0,C 180,E1 -20692.46,E2 -20692.46} C_VEL
LIN {X 0,Y 214.441,Z 323.761,A -85,B 0,C 180,E1 -20698.122,E2 -20698.122} C_VEL
LIN {X 0,Y 214.545,Z 323.751,A -85,B 0,C 180,E1 -20700,E2 -20700} C_VEL
LIN {X 0,Y 214.439,Z 323.769,A -85,B 0,C 180,E1 -20701.879,E2 -20701.879} C_VEL
LIN {X 0,Y 214.184,Z 323.801,A -85,B 0,C 180,E1 -20707.542,E2 -20707.542} C_VEL
LIN {X 0,Y 213.995,Z 323.812,A -85,B 0,C 180,E1 -20711.365,E2 -20711.365} C_VEL
LIN {X 0,Y 213.929,Z 323.829,A -85,B 0,C 180,E1 -20715.238,E2 -20715.238} C_VEL
LIN {X 0,Y 213.833,Z 323.844,A -85,B 0,C 180,E1 -20719.189,E2 -20719.189} C_VEL
LIN {X 0,Y 213.799,Z 323.841,A -85,B 0,C 180,E1 -20723.233,E2 -20723.233} C_VEL
LIN {X 0,Y 213.783,Z 323.843,A -85,B 0,C 180,E1 -20727.429,E2 -20727.429} C_VEL
LIN {X 0,Y 213.756,Z 323.856,A -85,B 0,C 180,E1 -20731.74,E2 -20731.74} C_VEL
LIN {X 0,Y 213.741,Z 323.857,A -85,B 0,C 180,E1 -20736.29,E2 -20736.29} C_VEL
LIN {X 0,Y 213.709,Z 323.853,A -85,B 0,C 180,E1 -20741.127,E2 -20741.127} C_VEL
LIN {X 0,Y 213.701,Z 323.861,A -85,B 0,C 180,E1 -20743.681,E2 -20743.681} C_VEL
LIN {X 0,Y 213.701,Z 323.864,A -85,B 0,C 180,E1 -20746.347,E2 -20746.347} C_VEL
LIN {X 0,Y 213.706,Z 323.862,A -85,B 0,C 180,E1 -20749.148,E2 -20749.148} C_VEL
LIN {X 0,Y 213.743,Z 323.853,A -85,B 0,C 180,E1 -20753.713,E2 -20753.713} C_VEL
LIN {X 0,Y 213.759,Z 323.856,A -85,B 0,C 180,E1 -20758.263,E2 -20758.263} C_VEL
LIN {X 0,Y 213.789,Z 323.853,A -85,B 0,C 180,E1 -20762.6,E2 -20762.6} C_VEL
LIN {X 0,Y 213.812,Z 323.85,A -85,B 0,C 180,E1 -20766.981,E2 -20766.981} C_VEL
LIN {X 0,Y 213.889,Z 323.84,A -85,B 0,C 180,E1 -20772.345,E2 -20772.345} C_VEL
LIN {X 0,Y 213.945,Z 323.832,A -85,B 0,C 180,E1 -20776.707,E2 -20776.707} C_VEL
LIN {X 0,Y 214.139,Z 323.808,A -85,B 0,C 180,E1 -20780.556,E2 -20780.556} C_VEL
LIN {X 0,Y 214.073,Z 323.82,A -85,B 0,C 180,E1 -20784.349,E2 -20784.349} C_VEL
LIN {X 0,Y 214.379,Z 323.784,A -85,B 0,C 180,E1 -20788.122,E2 -20788.122} C_VEL
LIN {X 0,Y 214.513,Z 323.766,A -85,B 0,C 180,E1 -20790.001,E2 -20790.001} C_VEL
LIN {X 0,Y 214.078,Z 323.82,A -85,B 0,C 180,E1 -20793.766,E2 -20793.766} C_VEL
LIN {X 0,Y 214.176,Z 323.806,A -85,B 0,C 180,E1 -20797.543,E2 -20797.543} C_VEL
LIN {X 0,Y 213.981,Z 323.829,A -85,B 0,C 180,E1 -20801.366,E2 -20801.366} C_VEL
LIN {X 0,Y 213.924,Z 323.994,A -85,B 0,C 180,E1 -20803.659,E2 -20803.659} C_VEL
LIN {X 0,Y 215.021,Z 326.86,A -85,B 0,C 180,E1 -20803.919,E2 -20803.919} C_VEL
LIN {X 0,Y 222.332,Z 343.729,A -85,B 0,C 180,E1 -20805.499,E2 -20805.499} C_VEL
LIN {X 0,Y 228.824,Z 362.065,A -85,B 0,C 180,E1 -20806.939,E2 -20806.939} C_VEL
LIN {X 0,Y 225.767,Z 428.058,A -85,B 0,C 180,E1 -20809.345,E2 -20809.345} C_VEL
LIN {X 0,Y 224.65,Z 441.672,A -85,B 0,C 180,E1 -20810.192,E2 -20810.192} C_VEL
LIN {X 0,Y 223.293,Z 454.721,A -85,B 0,C 180,E1 -20811.391,E2 -20811.391} C_VEL
LIN {X 0,Y 221.617,Z 467.117,A -85,B 0,C 180,E1 -20812.93,E2 -20812.93} C_VEL
LIN {X 0,Y 219.811,Z 478.716,A -85,B 0,C 180,E1 -20814.793,E2 -20814.793} C_VEL
LIN {X 0,Y 217.893,Z 489.913,A -85,B 0,C 180,E1 -20817.104,E2 -20817.104} C_VEL
LIN {X 0,Y 216.161,Z 499.059,A -85,B 0,C 180,E1 -20819.457,E2 -20819.457} C_VEL
LIN {X 0,Y 214.585,Z 507.516,A -85,B 0,C 180,E1 -20822.191,E2 -20822.191} C_VEL
LIN {X 0,Y 213.423,Z 513.541,A -85,B 0,C 180,E1 -20824.587,E2 -20824.587} C_VEL
LIN {X 0,Y 212.551,Z 519.363,A -85,B 0,C 180,E1 -20827.479,E2 -20827.479} C_VEL
LIN {X 0,Y 211.829,Z 523.748,A -85,B 0,C 180,E1 -20830.262,E2 -20830.262} C_VEL
LIN {X 0,Y 211.308,Z 526.996,A -85,B 0,C 180,E1 -20832.969,E2 -20832.969} C_VEL
LIN {X 0,Y 211.118,Z 529.315,A -85,B 0,C 180,E1 -20835.646,E2 -20835.646} C_VEL
LIN {X 0,Y 211.203,Z 530.761,A -85,B 0,C 180,E1 -20838.277,E2 -20838.277} C_VEL
LIN {X 0,Y 211.487,Z 531.41,A -85,B 0,C 180,E1 -20840.846,E2 -20840.846} C_VEL
LIN {X 0,Y 212.009,Z 531.365,A -85,B 0,C 180,E1 -20843.366,E2 -20843.366} C_VEL
LIN {X 0,Y 212.775,Z 530.622,A -85,B 0,C 180,E1 -20845.839,E2 -20845.839} C_VEL
LIN {X 0,Y 213.98,Z 528.926,A -85,B 0,C 180,E1 -20848.645,E2 -20848.645} C_VEL
LIN {X 0,Y 215.691,Z 526.093,A -85,B 0,C 180,E1 -20851.615,E2 -20851.615} C_VEL
LIN {X 0,Y 217.933,Z 522.088,A -85,B 0,C 180,E1 -20854.551,E2 -20854.551} C_VEL
LIN {X 0,Y 220.759,Z 516.57,A -85,B 0,C 180,E1 -20857.54,E2 -20857.54} C_VEL
LIN {X 0,Y 223.941,Z 509.869,A -85,B 0,C 180,E1 -20860.306,E2 -20860.306} C_VEL
LIN {X 0,Y 227.724,Z 501.175,A -85,B 0,C 180,E1 -20863.083,E2 -20863.083} C_VEL
LIN {X 0,Y 231.134,Z 492.499,A -85,B 0,C 180,E1 -20865.232,E2 -20865.232} C_VEL
LIN {X 0,Y 234.664,Z 482.268,A -85,B 0,C 180,E1 -20867.239,E2 -20867.239} C_VEL
LIN {X 0,Y 237.987,Z 471.241,A -85,B 0,C 180,E1 -20868.933,E2 -20868.933} C_VEL
LIN {X 0,Y 241.005,Z 459.275,A -85,B 0,C 180,E1 -20870.343,E2 -20870.343} C_VEL
LIN {X 0,Y 243.301,Z 447.269,A -85,B 0,C 180,E1 -20871.438,E2 -20871.438} C_VEL
LIN {X 0,Y 245.205,Z 434.594,A -85,B 0,C 180,E1 -20872.248,E2 -20872.248} C_VEL
LIN {X 0,Y 246.654,Z 419.068,A -85,B 0,C 180,E1 -20872.865,E2 -20872.865} C_VEL
LIN {X 0,Y 249.771,Z 377.871,A -85,B 0,C 180,E1 -20874.277,E2 -20874.277} C_VEL
LIN {X 0,Y 245.042,Z 367.666,A -85,B 0,C 180,E1 -20876.203,E2 -20876.203} C_VEL
LIN {X 0,Y 240.821,Z 359.823,A -85,B 0,C 180,E1 -20878.014,E2 -20878.014} C_VEL
LIN {X 0,Y 234.362,Z 349.326,A -85,B 0,C 180,E1 -20881.136,E2 -20881.136} C_VEL
LIN {X 0,Y 231.324,Z 345.032,A -85,B 0,C 180,E1 -20882.797,E2 -20882.797} C_VEL
LIN {X 0,Y 228.516,Z 341.497,A -85,B 0,C 180,E1 -20884.437,E2 -20884.437} C_VEL
LIN {X 0,Y 227.414,Z 340.352,A -85,B 0,C 180,E1 -20885.125,E2 -20885.125} C_VEL
LIN {X 0,Y 225.034,Z 337.809,A -85,B 0,C 180,E1 -20886.725,E2 -20886.725} C_VEL
LIN {X 0,Y 223.744,Z 335.439,A -85,B 0,C 180,E1 -20887.785,E2 -20887.785} C_VEL
LIN {X 0,Y 220.703,Z 332.773,A -85,B 0,C 180,E1 -20890.303,E2 -20890.303} C_VEL
LIN {X 0,Y 219.31,Z 330.617,A -85,B 0,C 180,E1 -20891.788,E2 -20891.788} C_VEL
LIN {X 0,Y 217.369,Z 329.042,A -85,B 0,C 180,E1 -20894.076,E2 -20894.076} C_VEL
LIN {X 0,Y 214.43,Z 325.94,A -85,B 0,C 180,E1 -20900.379,E2 -20900.379} C_VEL
LIN {X 0,Y 214.64,Z 326.365,A -85,B 0,C 180,E1 -20905.192,E2 -20905.192} C_VEL
LIN {X 0,Y 215.364,Z 327.607,A -85,B 0,C 180,E1 -20909.152,E2 -20909.152} C_VEL
LIN {X 0,Y 217.124,Z 330.799,A -85,B 0,C 180,E1 -20912.394,E2 -20912.394} C_VEL
LIN {X 0,Y 218.109,Z 332.935,A -85,B 0,C 180,E1 -20913.822,E2 -20913.822} C_VEL
LIN {X 0,Y 218.988,Z 336.045,A -85,B 0,C 180,E1 -20915.133,E2 -20915.133} C_VEL
LIN {X 0,Y 221.715,Z 345.483,A -85,B 0,C 180,E1 -20918.436,E2 -20918.436} C_VEL
LIN {X 0,Y 222.742,Z 347.374,A -85,B 0,C 180,E1 -20919.308,E2 -20919.308} C_VEL
LIN {X 0,Y 224.614,Z 350.074,A -85,B 0,C 180,E1 -20920.695,E2 -20920.695} C_VEL
LIN {X 0,Y 228.267,Z 355.909,A -85,B 0,C 180,E1 -20923.113,E2 -20923.113} C_VEL
LIN {X 0,Y 231.421,Z 361.413,A -85,B 0,C 180,E1 -20924.991,E2 -20924.991} C_VEL
LIN {X 0,Y 234.418,Z 366.878,A -85,B 0,C 180,E1 -20926.585,E2 -20926.585} C_VEL
LIN {X 0,Y 238.076,Z 374.299,A -85,B 0,C 180,E1 -20928.424,E2 -20928.424} C_VEL
LIN {X 0,Y 242.319,Z 384.305,A -85,B 0,C 180,E1 -20930.397,E2 -20930.397} C_VEL
LIN {X 0,Y 243.558,Z 388.107,A -85,B 0,C 180,E1 -20930.997,E2 -20930.997} C_VEL
LIN {X 0,Y 244.066,Z 395.828,A -85,B 0,C 180,E1 -20931.598,E2 -20931.598} C_VEL
LIN {X 0,Y 240.195,Z 442.326,A -85,B 0,C 180,E1 -20933.225,E2 -20933.225} C_VEL
LIN {X 0,Y 238.156,Z 455.8,A -85,B 0,C 180,E1 -20933.959,E2 -20933.959} C_VEL
LIN {X 0,Y 235.506,Z 468.311,A -85,B 0,C 180,E1 -20934.937,E2 -20934.937} C_VEL
LIN {X 0,Y 232.269,Z 480.344,A -85,B 0,C 180,E1 -20936.22,E2 -20936.22} C_VEL
LIN {X 0,Y 228.817,Z 491.275,A -85,B 0,C 180,E1 -20937.746,E2 -20937.746} C_VEL
LIN {X 0,Y 225.571,Z 500.251,A -85,B 0,C 180,E1 -20939.323,E2 -20939.323} C_VEL
LIN {X 0,Y 221.447,Z 510.45,A -85,B 0,C 180,E1 -20941.571,E2 -20941.571} C_VEL
LIN {X 0,Y 217.592,Z 519.432,A -85,B 0,C 180,E1 -20944.148,E2 -20944.148} C_VEL
LIN {X 0,Y 214.096,Z 526.747,A -85,B 0,C 180,E1 -20946.801,E2 -20946.801} C_VEL
LIN {X 0,Y 211.329,Z 532.646,A -85,B 0,C 180,E1 -20949.561,E2 -20949.561} C_VEL
LIN {X 0,Y 208.826,Z 537.358,A -85,B 0,C 180,E1 -20952.367,E2 -20952.367} C_VEL
LIN {X 0,Y 206.868,Z 541.011,A -85,B 0,C 180,E1 -20955.237,E2 -20955.237} C_VEL
LIN {X 0,Y 205.616,Z 543.675,A -85,B 0,C 180,E1 -20958.165,E2 -20958.165} C_VEL
LIN {X 0,Y 205.052,Z 544.96,A -85,B 0,C 180,E1 -20960.131,E2 -20960.131} C_VEL
LIN {X 0,Y 204.402,Z 546.265,A -85,B 0,C 180,E1 -20964.078,E2 -20964.078} C_VEL
LIN {X 0,Y 204.364,Z 546.338,A -85,B 0,C 180,E1 -20966.055,E2 -20966.055} C_VEL
LIN {X 0,Y 204.461,Z 546.023,A -85,B 0,C 180,E1 -20968.029,E2 -20968.029} C_VEL
LIN {X 0,Y 204.618,Z 545.269,A -85,B 0,C 180,E1 -20969.999,E2 -20969.999} C_VEL
LIN {X 0,Y 204.524,Z 544.059,A -85,B 0,C 180,E1 -20971.968,E2 -20971.968} C_VEL
LIN {X 0,Y 204.53,Z 541.559,A -85,B 0,C 180,E1 -20974.804,E2 -20974.804} C_VEL
LIN {X 0,Y 204.711,Z 537.702,A -85,B 0,C 180,E1 -20977.892,E2 -20977.892} C_VEL
LIN {X 0,Y 205.21,Z 532.79,A -85,B 0,C 180,E1 -20980.856,E2 -20980.856} C_VEL
LIN {X 0,Y 206.102,Z 526.544,A -85,B 0,C 180,E1 -20983.808,E2 -20983.808} C_VEL
LIN {X 0,Y 207.555,Z 518.749,A -85,B 0,C 180,E1 -20986.726,E2 -20986.726} C_VEL
LIN {X 0,Y 209.029,Z 510.711,A -85,B 0,C 180,E1 -20989.135,E2 -20989.135} C_VEL
LIN {X 0,Y 210.92,Z 500.917,A -85,B 0,C 180,E1 -20991.5,E2 -20991.5} C_VEL
LIN {X 0,Y 212.868,Z 490.056,A -85,B 0,C 180,E1 -20993.597,E2 -20993.597} C_VEL
LIN {X 0,Y 214.617,Z 479.55,A -85,B 0,C 180,E1 -20995.194,E2 -20995.194} C_VEL
LIN {X 0,Y 216.408,Z 467.074,A -85,B 0,C 180,E1 -20996.651,E2 -20996.651} C_VEL
LIN {X 0,Y 217.944,Z 454.252,A -85,B 0,C 180,E1 -20997.745,E2 -20997.745} C_VEL
LIN {X 0,Y 218.925,Z 441.94,A -85,B 0,C 180,E1 -20998.457,E2 -20998.457} C_VEL
LIN {X 0,Y 221.302,Z 388.969,A -85,B 0,C 180,E1 -21000.451,E2 -21000.451} C_VEL
LIN {X 0,Y 217.611,Z 359.014,A -85,B 0,C 180,E1 -21002.116,E2 -21002.116} C_VEL
LIN {X 0,Y 208.928,Z 334.807,A -85,B 0,C 180,E1 -21004.262,E2 -21004.262} C_VEL
LIN {X 0,Y 206.914,Z 325.423,A -85,B 0,C 180,E1 -21008.629,E2 -21008.629} C_VEL
LIN {X 0,Y 206.741,Z 324.736,A -85,B 0,C 180,E1 -21008.99,E2 -21008.99} C_VEL
LIN {X 0,Y 206.627,Z 324.748,A -85,B 0,C 180,E1 -21014.417,E2 -21014.417} C_VEL
LIN {X 0,Y 206.661,Z 324.742,A -85,B 0,C 180,E1 -21019.749,E2 -21019.749} C_VEL
LIN {X 0,Y 206.727,Z 324.736,A -85,B 0,C 180,E1 -21024.695,E2 -21024.695} C_VEL
LIN {X 0,Y 206.719,Z 324.713,A -85,B 0,C 180,E1 -21029.339,E2 -21029.339} C_VEL
LIN {X 0,Y 206.729,Z 324.733,A -85,B 0,C 180,E1 -21033.772,E2 -21033.772} C_VEL
LIN {X 0,Y 206.753,Z 324.728,A -85,B 0,C 180,E1 -21038.043,E2 -21038.043} C_VEL
LIN {X 0,Y 206.869,Z 324.715,A -85,B 0,C 180,E1 -21042.197,E2 -21042.197} C_VEL
LIN {X 0,Y 206.909,Z 324.706,A -85,B 0,C 180,E1 -21046.246,E2 -21046.246} C_VEL
LIN {X 0,Y 207.101,Z 324.683,A -85,B 0,C 180,E1 -21050.231,E2 -21050.231} C_VEL
LIN {X 0,Y 207.164,Z 324.678,A -85,B 0,C 180,E1 -21052.201,E2 -21052.201} C_VEL
LIN {X 0,Y 207.377,Z 324.64,A -85,B 0,C 180,E1 -21058.058,E2 -21058.058} C_VEL
LIN {X 0,Y 207.51,Z 324.626,A -85,B 0,C 180,E1 -21060,E2 -21060} C_VEL
LIN {X 0,Y 207.376,Z 324.649,A -85,B 0,C 180,E1 -21061.943,E2 -21061.943} C_VEL
LIN {X 0,Y 207.128,Z 324.679,A -85,B 0,C 180,E1 -21067.801,E2 -21067.801} C_VEL
LIN {X 0,Y 206.92,Z 324.692,A -85,B 0,C 180,E1 -21071.759,E2 -21071.759} C_VEL
LIN {X 0,Y 206.863,Z 324.71,A -85,B 0,C 180,E1 -21075.772,E2 -21075.772} C_VEL
LIN {X 0,Y 206.776,Z 324.725,A -85,B 0,C 180,E1 -21079.87,E2 -21079.87} C_VEL
LIN {X 0,Y 206.734,Z 324.719,A -85,B 0,C 180,E1 -21084.076,E2 -21084.076} C_VEL
LIN {X 0,Y 206.685,Z 324.73,A -85,B 0,C 180,E1 -21088.428,E2 -21088.428} C_VEL
LIN {X 0,Y 206.692,Z 324.738,A -85,B 0,C 180,E1 -21092.96,E2 -21092.96} C_VEL
LIN {X 0,Y 206.677,Z 324.73,A -85,B 0,C 180,E1 -21097.741,E2 -21097.741} C_VEL
LIN {X 0,Y 206.639,Z 324.735,A -85,B 0,C 180,E1 -21101.564,E2 -21101.564} C_VEL
LIN {X 0,Y 206.629,Z 324.745,A -85,B 0,C 180,E1 -21105.584,E2 -21105.584} C_VEL
LIN {X 0,Y 206.649,Z 324.738,A -85,B 0,C 180,E1 -21109.748,E2 -21109.748} C_VEL
LIN {X 0,Y 206.699,Z 324.73,A -85,B 0,C 180,E1 -21114.69,E2 -21114.69} C_VEL
LIN {X 0,Y 206.696,Z 324.738,A -85,B 0,C 180,E1 -21119.336,E2 -21119.336} C_VEL
LIN {X 0,Y 206.706,Z 324.736,A -85,B 0,C 180,E1 -21123.77,E2 -21123.77} C_VEL
LIN {X 0,Y 206.735,Z 324.732,A -85,B 0,C 180,E1 -21128.042,E2 -21128.042} C_VEL
LIN {X 0,Y 206.829,Z 324.72,A -85,B 0,C 180,E1 -21132.194,E2 -21132.194} C_VEL
LIN {X 0,Y 206.885,Z 324.713,A -85,B 0,C 180,E1 -21136.245,E2 -21136.245} C_VEL
LIN {X 0,Y 207.083,Z 324.688,A -85,B 0,C 180,E1 -21140.231,E2 -21140.231} C_VEL
LIN {X 0,Y 207.037,Z 324.696,A -85,B 0,C 180,E1 -21144.156,E2 -21144.156} C_VEL
LIN {X 0,Y 207.321,Z 324.663,A -85,B 0,C 180,E1 -21148.059,E2 -21148.059} C_VEL
LIN {X 0,Y 207.481,Z 324.642,A -85,B 0,C 180,E1 -21150.001,E2 -21150.001} C_VEL
LIN {X 0,Y 207.024,Z 324.7,A -85,B 0,C 180,E1 -21153.894,E2 -21153.894} C_VEL
LIN {X 0,Y 207.121,Z 324.686,A -85,B 0,C 180,E1 -21157.802,E2 -21157.802} C_VEL
LIN {X 0,Y 206.903,Z 324.711,A -85,B 0,C 180,E1 -21161.761,E2 -21161.761} C_VEL
LIN {X 0,Y 206.89,Z 324.811,A -85,B 0,C 180,E1 -21162.795,E2 -21162.795} C_VEL
LIN {X 0,Y 207.978,Z 327.715,A -85,B 0,C 180,E1 -21163.069,E2 -21163.069} C_VEL
LIN {X 0,Y 216.164,Z 346.364,A -85,B 0,C 180,E1 -21164.907,E2 -21164.907} C_VEL
LIN {X 0,Y 222.162,Z 363.503,A -85,B 0,C 180,E1 -21166.306,E2 -21166.306} C_VEL
LIN {X 0,Y 219.082,Z 428.229,A -85,B 0,C 180,E1 -21168.741,E2 -21168.741} C_VEL
LIN {X 0,Y 217.957,Z 441.446,A -85,B 0,C 180,E1 -21169.579,E2 -21169.579} C_VEL
LIN {X 0,Y 216.679,Z 453.868,A -85,B 0,C 180,E1 -21170.727,E2 -21170.727} C_VEL
LIN {X 0,Y 215.05,Z 465.762,A -85,B 0,C 180,E1 -21172.203,E2 -21172.203} C_VEL
LIN {X 0,Y 213.164,Z 477.484,A -85,B 0,C 180,E1 -21174.08,E2 -21174.08} C_VEL
LIN {X 0,Y 211.414,Z 487.736,A -85,B 0,C 180,E1 -21176.16,E2 -21176.16} C_VEL
LIN {X 0,Y 209.594,Z 497.113,A -85,B 0,C 180,E1 -21178.532,E2 -21178.532} C_VEL
LIN {X 0,Y 208.023,Z 505.078,A -85,B 0,C 180,E1 -21181.013,E2 -21181.013} C_VEL
LIN {X 0,Y 206.57,Z 512.755,A -85,B 0,C 180,E1 -21183.985,E2 -21183.985} C_VEL
LIN {X 0,Y 205.628,Z 518.394,A -85,B 0,C 180,E1 -21186.736,E2 -21186.736} C_VEL
LIN {X 0,Y 204.946,Z 522.705,A -85,B 0,C 180,E1 -21189.375,E2 -21189.375} C_VEL
LIN {X 0,Y 204.315,Z 526.232,A -85,B 0,C 180,E1 -21192.138,E2 -21192.138} C_VEL
LIN {X 0,Y 204.033,Z 528.974,A -85,B 0,C 180,E1 -21195.079,E2 -21195.079} C_VEL
LIN {X 0,Y 204.037,Z 529.927,A -85,B 0,C 180,E1 -21196.456,E2 -21196.456} C_VEL
LIN {X 0,Y 204.196,Z 531.241,A -85,B 0,C 180,E1 -21199.219,E2 -21199.219} C_VEL
LIN {X 0,Y 204.609,Z 531.776,A -85,B 0,C 180,E1 -21202.188,E2 -21202.188} C_VEL
LIN {X 0,Y 205.424,Z 531.379,A -85,B 0,C 180,E1 -21205.195,E2 -21205.195} C_VEL
LIN {X 0,Y 206.646,Z 530.002,A -85,B 0,C 180,E1 -21208.24,E2 -21208.24} C_VEL
LIN {X 0,Y 208.69,Z 526.978,A -85,B 0,C 180,E1 -21211.869,E2 -21211.869} C_VEL
LIN {X 0,Y 211.518,Z 522.345,A -85,B 0,C 180,E1 -21215.483,E2 -21215.483} C_VEL
LIN {X 0,Y 214.122,Z 517.678,A -85,B 0,C 180,E1 -21218.127,E2 -21218.127} C_VEL
LIN {X 0,Y 217.115,Z 511.874,A -85,B 0,C 180,E1 -21220.707,E2 -21220.707} C_VEL
LIN {X 0,Y 220.704,Z 504.292,A -85,B 0,C 180,E1 -21223.345,E2 -21223.345} C_VEL
LIN {X 0,Y 224.676,Z 494.973,A -85,B 0,C 180,E1 -21225.862,E2 -21225.862} C_VEL
LIN {X 0,Y 228.23,Z 485.772,A -85,B 0,C 180,E1 -21227.822,E2 -21227.822} C_VEL
LIN {X 0,Y 231.511,Z 475.919,A -85,B 0,C 180,E1 -21229.505,E2 -21229.505} C_VEL
LIN {X 0,Y 234.812,Z 464.472,A -85,B 0,C 180,E1 -21231.008,E2 -21231.008} C_VEL
LIN {X 0,Y 237.526,Z 452.449,A -85,B 0,C 180,E1 -21232.241,E2 -21232.241} C_VEL
LIN {X 0,Y 239.64,Z 440.055,A -85,B 0,C 180,E1 -21233.183,E2 -21233.183} C_VEL
LIN {X 0,Y 241.281,Z 426.206,A -85,B 0,C 180,E1 -21233.865,E2 -21233.865} C_VEL
LIN {X 0,Y 245.059,Z 380.92,A -85,B 0,C 180,E1 -21235.409,E2 -21235.409} C_VEL
LIN {X 0,Y 241.056,Z 371.997,A -85,B 0,C 180,E1 -21237.176,E2 -21237.176} C_VEL
LIN {X 0,Y 237.215,Z 364.514,A -85,B 0,C 180,E1 -21238.97,E2 -21238.97} C_VEL
LIN {X 0,Y 231.223,Z 354.717,A -85,B 0,C 180,E1 -21242.057,E2 -21242.057} C_VEL
LIN {X 0,Y 228.692,Z 351.049,A -85,B 0,C 180,E1 -21243.523,E2 -21243.523} C_VEL
LIN {X 0,Y 225.78,Z 347.207,A -85,B 0,C 180,E1 -21245.358,E2 -21245.358} C_VEL
LIN {X 0,Y 223.145,Z 344.49,A -85,B 0,C 180,E1 -21247.173,E2 -21247.173} C_VEL
LIN {X 0,Y 221.745,Z 341.954,A -85,B 0,C 180,E1 -21248.371,E2 -21248.371} C_VEL
LIN {X 0,Y 219.009,Z 339.425,A -85,B 0,C 180,E1 -21250.775,E2 -21250.775} C_VEL
LIN {X 0,Y 217.734,Z 337.346,A -85,B 0,C 180,E1 -21252.229,E2 -21252.229} C_VEL
LIN {X 0,Y 215.724,Z 335.773,A -85,B 0,C 180,E1 -21254.718,E2 -21254.718} C_VEL
LIN {X 0,Y 213.291,Z 332.98,A -85,B 0,C 180,E1 -21260.241,E2 -21260.241} C_VEL
LIN {X 0,Y 212.942,Z 333.149,A -85,B 0,C 180,E1 -21264.365,E2 -21264.365} C_VEL
LIN {X 0,Y 214.059,Z 334.449,A -85,B 0,C 180,E1 -21268.776,E2 -21268.776} C_VEL
LIN {X 0,Y 218.133,Z 340.747,A -85,B 0,C 180,E1 -21275.085,E2 -21275.085} C_VEL
LIN {X 0,Y 219.824,Z 342.832,A -85,B 0,C 180,E1 -21276.759,E2 -21276.759} C_VEL
LIN {X 0,Y 222.742,Z 347.374,A -85,B 0,C 180,E1 -21279.308,E2 -21279.308} C_VEL
LIN {X 0,Y 224.244,Z 350.544,A -85,B 0,C 180,E1 -21280.521,E2 -21280.521} C_VEL
LIN {X 0,Y 225.432,Z 354.667,A -85,B 0,C 180,E1 -21281.57,E2 -21281.57} C_VEL
LIN {X 0,Y 227.622,Z 363.824,A -85,B 0,C 180,E1 -21283.474,E2 -21283.474} C_VEL
LIN {X 0,Y 229.102,Z 367.992,A -85,B 0,C 180,E1 -21284.496,E2 -21284.496} C_VEL
LIN {X 0,Y 229.716,Z 369.2,A -85,B 0,C 180,E1 -21284.865,E2 -21284.865} C_VEL
LIN {X 0,Y 234.034,Z 377.873,A -85,B 0,C 180,E1 -21287.212,E2 -21287.212} C_VEL
LIN {X 0,Y 238.237,Z 388.163,A -85,B 0,C 180,E1 -21289.356,E2 -21289.356} C_VEL
LIN {X 0,Y 239.244,Z 391.417,A -85,B 0,C 180,E1 -21289.879,E2 -21289.879} C_VEL
LIN {X 0,Y 239.555,Z 397.05,A -85,B 0,C 180,E1 -21290.322,E2 -21290.322} C_VEL
LIN {X 0,Y 235.545,Z 442.246,A -85,B 0,C 180,E1 -21291.938,E2 -21291.938} C_VEL
LIN {X 0,Y 233.301,Z 456.097,A -85,B 0,C 180,E1 -21292.702,E2 -21292.702} C_VEL
LIN {X 0,Y 230.344,Z 469.158,A -85,B 0,C 180,E1 -21293.761,E2 -21293.761} C_VEL
LIN {X 0,Y 226.973,Z 480.984,A -85,B 0,C 180,E1 -21295.051,E2 -21295.051} C_VEL
LIN {X 0,Y 223.375,Z 491.761,A -85,B 0,C 180,E1 -21296.591,E2 -21296.591} C_VEL
LIN {X 0,Y 219.976,Z 500.619,A -85,B 0,C 180,E1 -21298.185,E2 -21298.185} C_VEL
LIN {X 0,Y 216.114,Z 509.81,A -85,B 0,C 180,E1 -21300.268,E2 -21300.268} C_VEL
LIN {X 0,Y 212.551,Z 517.459,A -85,B 0,C 180,E1 -21302.424,E2 -21302.424} C_VEL
LIN {X 0,Y 208.175,Z 526.163,A -85,B 0,C 180,E1 -21305.57,E2 -21305.57} C_VEL
LIN {X 0,Y 205.534,Z 531.206,A -85,B 0,C 180,E1 -21307.905,E2 -21307.905} C_VEL
LIN {X 0,Y 202.913,Z 536.149,A -85,B 0,C 180,E1 -21310.789,E2 -21310.789} C_VEL
LIN {X 0,Y 200.597,Z 540.011,A -85,B 0,C 180,E1 -21313.722,E2 -21313.722} C_VEL
LIN {X 0,Y 198.636,Z 543.646,A -85,B 0,C 180,E1 -21317.742,E2 -21317.742} C_VEL
LIN {X 0,Y 198.025,Z 544.83,A -85,B 0,C 180,E1 -21319.777,E2 -21319.777} C_VEL
LIN {X 0,Y 197.34,Z 546.02,A -85,B 0,C 180,E1 -21323.866,E2 -21323.866} C_VEL
LIN {X 0,Y 197.285,Z 546.038,A -85,B 0,C 180,E1 -21325.913,E2 -21325.913} C_VEL
LIN {X 0,Y 197.378,Z 545.636,A -85,B 0,C 180,E1 -21327.958,E2 -21327.958} C_VEL
LIN {X 0,Y 197.553,Z 544.809,A -85,B 0,C 180,E1 -21329.999,E2 -21329.999} C_VEL
LIN {X 0,Y 197.442,Z 543.548,A -85,B 0,C 180,E1 -21332.039,E2 -21332.039} C_VEL
LIN {X 0,Y 197.431,Z 541.294,A -85,B 0,C 180,E1 -21334.64,E2 -21334.64} C_VEL
LIN {X 0,Y 197.661,Z 536.974,A -85,B 0,C 180,E1 -21338.175,E2 -21338.175} C_VEL
LIN {X 0,Y 198.193,Z 531.944,A -85,B 0,C 180,E1 -21341.245,E2 -21341.245} C_VEL
LIN {X 0,Y 199.182,Z 525.565,A -85,B 0,C 180,E1 -21344.298,E2 -21344.298} C_VEL
LIN {X 0,Y 200.69,Z 517.53,A -85,B 0,C 180,E1 -21347.316,E2 -21347.316} C_VEL
LIN {X 0,Y 202.23,Z 509.293,A -85,B 0,C 180,E1 -21349.805,E2 -21349.805} C_VEL
LIN {X 0,Y 204.255,Z 499.278,A -85,B 0,C 180,E1 -21352.239,E2 -21352.239} C_VEL
LIN {X 0,Y 206.086,Z 489.439,A -85,B 0,C 180,E1 -21354.155,E2 -21354.155} C_VEL
LIN {X 0,Y 207.904,Z 478.826,A -85,B 0,C 180,E1 -21355.798,E2 -21355.798} C_VEL
LIN {X 0,Y 209.731,Z 466.222,A -85,B 0,C 180,E1 -21357.299,E2 -21357.299} C_VEL
LIN {X 0,Y 211.288,Z 453.128,A -85,B 0,C 180,E1 -21358.428,E2 -21358.428} C_VEL
LIN {X 0,Y 212.327,Z 440.319,A -85,B 0,C 180,E1 -21359.155,E2 -21359.155} C_VEL
LIN {X 0,Y 214.644,Z 389.301,A -85,B 0,C 180,E1 -21361.133,E2 -21361.133} C_VEL
LIN {X 0,Y 211.387,Z 361.607,A -85,B 0,C 180,E1 -21362.723,E2 -21362.723} C_VEL
LIN {X 0,Y 202.648,Z 337.44,A -85,B 0,C 180,E1 -21364.912,E2 -21364.912} C_VEL
LIN {X 0,Y 201.668,Z 334.635,A -85,B 0,C 180,E1 -21365.181,E2 -21365.181} C_VEL
LIN {X 0,Y 199.683,Z 325.615,A -85,B 0,C 180,E1 -21369.602,E2 -21369.602} C_VEL
LIN {X 0,Y 199.573,Z 325.625,A -85,B 0,C 180,E1 -21375.227,E2 -21375.227} C_VEL
LIN {X 0,Y 199.635,Z 325.62,A -85,B 0,C 180,E1 -21380.678,E2 -21380.678} C_VEL
LIN {X 0,Y 199.631,Z 325.615,A -85,B 0,C 180,E1 -21385.717,E2 -21385.717} C_VEL
LIN {X 0,Y 199.7,Z 325.597,A -85,B 0,C 180,E1 -21388.137,E2 -21388.137} C_VEL
LIN {X 0,Y 199.683,Z 325.607,A -85,B 0,C 180,E1 -21392.771,E2 -21392.771} C_VEL
LIN {X 0,Y 199.733,Z 325.606,A -85,B 0,C 180,E1 -21397.229,E2 -21397.229} C_VEL
LIN {X 0,Y 199.792,Z 325.597,A -85,B 0,C 180,E1 -21401.757,E2 -21401.757} C_VEL
LIN {X 0,Y 199.843,Z 325.588,A -85,B 0,C 180,E1 -21405.749,E2 -21405.749} C_VEL
LIN {X 0,Y 200.066,Z 325.56,A -85,B 0,C 180,E1 -21409.884,E2 -21409.884} C_VEL
LIN {X 0,Y 200.03,Z 325.567,A -85,B 0,C 180,E1 -21413.95,E2 -21413.95} C_VEL
LIN {X 0,Y 200.317,Z 325.519,A -85,B 0,C 180,E1 -21417.99,E2 -21417.99} C_VEL
LIN {X 0,Y 200.474,Z 325.501,A -85,B 0,C 180,E1 -21420,E2 -21420} C_VEL
LIN {X 0,Y 200.018,Z 325.568,A -85,B 0,C 180,E1 -21424.03,E2 -21424.03} C_VEL
LIN {X 0,Y 200.075,Z 325.555,A -85,B 0,C 180,E1 -21428.078,E2 -21428.078} C_VEL
LIN {X 0,Y 199.87,Z 325.571,A -85,B 0,C 180,E1 -21432.18,E2 -21432.18} C_VEL
LIN {X 0,Y 199.801,Z 325.594,A -85,B 0,C 180,E1 -21436.344,E2 -21436.344} C_VEL
LIN {X 0,Y 199.687,Z 325.605,A -85,B 0,C 180,E1 -21440.607,E2 -21440.607} C_VEL
LIN {X 0,Y 199.647,Z 325.594,A -85,B 0,C 180,E1 -21444.989,E2 -21444.989} C_VEL
LIN {X 0,Y 199.605,Z 325.615,A -85,B 0,C 180,E1 -21449.534,E2 -21449.534} C_VEL
LIN {X 0,Y 199.663,Z 325.614,A -85,B 0,C 180,E1 -21452.354,E2 -21452.354} C_VEL
LIN {X 0,Y 199.621,Z 325.613,A -85,B 0,C 180,E1 -21456.765,E2 -21456.765} C_VEL
LIN {X 0,Y 199.605,Z 325.603,A -85,B 0,C 180,E1 -21459.33,E2 -21459.33} C_VEL
LIN {X 0,Y 199.57,Z 325.615,A -85,B 0,C 180,E1 -21462.311,E2 -21462.311} C_VEL
LIN {X 0,Y 199.576,Z 325.625,A -85,B 0,C 180,E1 -21465.23,E2 -21465.23} C_VEL
LIN {X 0,Y 199.572,Z 325.623,A -85,B 0,C 180,E1 -21468.005,E2 -21468.005} C_VEL
LIN {X 0,Y 199.599,Z 325.615,A -85,B 0,C 180,E1 -21470.773,E2 -21470.773} C_VEL
LIN {X 0,Y 199.613,Z 325.611,A -85,B 0,C 180,E1 -21474.077,E2 -21474.077} C_VEL
LIN {X 0,Y 199.686,Z 325.61,A -85,B 0,C 180,E1 -21478.136,E2 -21478.136} C_VEL
LIN {X 0,Y 199.644,Z 325.615,A -85,B 0,C 180,E1 -21482.767,E2 -21482.767} C_VEL
LIN {X 0,Y 199.709,Z 325.608,A -85,B 0,C 180,E1 -21487.227,E2 -21487.227} C_VEL
LIN {X 0,Y 199.753,Z 325.603,A -85,B 0,C 180,E1 -21491.799,E2 -21491.799} C_VEL
LIN {X 0,Y 199.821,Z 325.595,A -85,B 0,C 180,E1 -21495.749,E2 -21495.749} C_VEL
LIN {X 0,Y 200.026,Z 325.57,A -85,B 0,C 180,E1 -21499.883,E2 -21499.883} C_VEL
LIN {X 0,Y 200.002,Z 325.573,A -85,B 0,C 180,E1 -21503.95,E2 -21503.95} C_VEL
LIN {X 0,Y 200.266,Z 325.541,A -85,B 0,C 180,E1 -21507.99,E2 -21507.99} C_VEL
LIN {X 0,Y 200.447,Z 325.518,A -85,B 0,C 180,E1 -21510.001,E2 -21510.001} C_VEL
LIN {X 0,Y 199.972,Z 325.579,A -85,B 0,C 180,E1 -21514.032,E2 -21514.032} C_VEL
LIN {X 0,Y 200.07,Z 325.565,A -85,B 0,C 180,E1 -21518.079,E2 -21518.079} C_VEL
LIN {X 0,Y 199.866,Z 325.587,A -85,B 0,C 180,E1 -21521.859,E2 -21521.859} C_VEL
LIN {X 0,Y 200.898,Z 328.47,A -85,B 0,C 180,E1 -21522.171,E2 -21522.171} C_VEL
LIN {X 0,Y 209.582,Z 348.036,A -85,B 0,C 180,E1 -21524.195,E2 -21524.195} C_VEL
LIN {X 0,Y 215.552,Z 365.015,A -85,B 0,C 180,E1 -21525.645,E2 -21525.645} C_VEL
LIN {X 0,Y 212.36,Z 429.117,A -85,B 0,C 180,E1 -21528.138,E2 -21528.138} C_VEL
LIN {X 0,Y 211.244,Z 441.999,A -85,B 0,C 180,E1 -21528.992,E2 -21528.992} C_VEL
LIN {X 0,Y 209.919,Z 454.128,A -85,B 0,C 180,E1 -21530.147,E2 -21530.147} C_VEL
LIN {X 0,Y 208.054,Z 467.034,A -85,B 0,C 180,E1 -21531.814,E2 -21531.814} C_VEL
LIN {X 0,Y 206.219,Z 478.215,A -85,B 0,C 180,E1 -21533.687,E2 -21533.687} C_VEL
LIN {X 0,Y 204.358,Z 488.595,A -85,B 0,C 180,E1 -21535.891,E2 -21535.891} C_VEL
LIN {X 0,Y 202.386,Z 498.469,A -85,B 0,C 180,E1 -21538.522,E2 -21538.522} C_VEL
LIN {X 0,Y 200.818,Z 506.312,A -85,B 0,C 180,E1 -21541.116,E2 -21541.116} C_VEL
LIN {X 0,Y 199.47,Z 513.061,A -85,B 0,C 180,E1 -21543.865,E2 -21543.865} C_VEL
LIN {X 0,Y 198.449,Z 519.207,A -85,B 0,C 180,E1 -21547.018,E2 -21547.018} C_VEL
LIN {X 0,Y 197.732,Z 523.458,A -85,B 0,C 180,E1 -21549.776,E2 -21549.776} C_VEL
LIN {X 0,Y 197.145,Z 526.865,A -85,B 0,C 180,E1 -21552.637,E2 -21552.637} C_VEL
LIN {X 0,Y 196.927,Z 529.394,A -85,B 0,C 180,E1 -21555.544,E2 -21555.544} C_VEL
LIN {X 0,Y 197.013,Z 531.094,A -85,B 0,C 180,E1 -21558.516,E2 -21558.516} C_VEL
LIN {X 0,Y 197.382,Z 531.951,A -85,B 0,C 180,E1 -21561.568,E2 -21561.568} C_VEL
LIN {X 0,Y 198.397,Z 531.745,A -85,B 0,C 180,E1 -21565.473,E2 -21565.473} C_VEL
LIN {X 0,Y 199.447,Z 530.761,A -85,B 0,C 180,E1 -21568.091,E2 -21568.091} C_VEL
LIN {X 0,Y 201.681,Z 527.95,A -85,B 0,C 180,E1 -21572.066,E2 -21572.066} C_VEL
LIN {X 0,Y 204.421,Z 523.828,A -85,B 0,C 180,E1 -21575.634,E2 -21575.634} C_VEL
LIN {X 0,Y 207.377,Z 518.982,A -85,B 0,C 180,E1 -21578.63,E2 -21578.63} C_VEL
LIN {X 0,Y 210.8,Z 512.82,A -85,B 0,C 180,E1 -21581.534,E2 -21581.534} C_VEL
LIN {X 0,Y 214.24,Z 506.134,A -85,B 0,C 180,E1 -21584.008,E2 -21584.008} C_VEL
LIN {X 0,Y 218.202,Z 497.624,A -85,B 0,C 180,E1 -21586.499,E2 -21586.499} C_VEL
LIN {X 0,Y 222.199,Z 488.018,A -85,B 0,C 180,E1 -21588.672,E2 -21588.672} C_VEL
LIN {X 0,Y 226.098,Z 477.14,A -85,B 0,C 180,E1 -21590.607,E2 -21590.607} C_VEL
LIN {X 0,Y 229.436,Z 466.386,A -85,B 0,C 180,E1 -21592.077,E2 -21592.077} C_VEL
LIN {X 0,Y 232.241,Z 454.959,A -85,B 0,C 180,E1 -21593.314,E2 -21593.314} C_VEL
LIN {X 0,Y 234.646,Z 442.139,A -85,B 0,C 180,E1 -21594.36,E2 -21594.36} C_VEL
LIN {X 0,Y 236.503,Z 428.755,A -85,B 0,C 180,E1 -21595.065,E2 -21595.065} C_VEL
LIN {X 0,Y 240.364,Z 383.41,A -85,B 0,C 180,E1 -21596.683,E2 -21596.683} C_VEL
LIN {X 0,Y 235.543,Z 372.786,A -85,B 0,C 180,E1 -21599.009,E2 -21599.009} C_VEL
LIN {X 0,Y 230.978,Z 364.878,A -85,B 0,C 180,E1 -21601.358,E2 -21601.358} C_VEL
LIN {X 0,Y 228.433,Z 360.456,A -85,B 0,C 180,E1 -21602.854,E2 -21602.854} C_VEL
LIN {X 0,Y 226.282,Z 357.239,A -85,B 0,C 180,E1 -21604.16,E2 -21604.16} C_VEL
LIN {X 0,Y 223.457,Z 353.52,A -85,B 0,C 180,E1 -21606.056,E2 -21606.056} C_VEL
LIN {X 0,Y 220.837,Z 350.438,A -85,B 0,C 180,E1 -21608.003,E2 -21608.003} C_VEL
LIN {X 0,Y 219.855,Z 348.602,A -85,B 0,C 180,E1 -21608.912,E2 -21608.912} C_VEL
LIN {X 0,Y 217.225,Z 345.918,A -85,B 0,C 180,E1 -21611.37,E2 -21611.37} C_VEL
LIN {X 0,Y 216.03,Z 343.969,A -85,B 0,C 180,E1 -21612.846,E2 -21612.846} C_VEL
LIN {X 0,Y 212.857,Z 341.158,A -85,B 0,C 180,E1 -21617.879,E2 -21617.879} C_VEL
LIN {X 0,Y 212.136,Z 339.983,A -85,B 0,C 180,E1 -21620.356,E2 -21620.356} C_VEL
LIN {X 0,Y 211.879,Z 340.279,A -85,B 0,C 180,E1 -21625.019,E2 -21625.019} C_VEL
LIN {X 0,Y 212.876,Z 341.559,A -85,B 0,C 180,E1 -21628.708,E2 -21628.708} C_VEL
LIN {X 0,Y 216.581,Z 347.541,A -85,B 0,C 180,E1 -21634.715,E2 -21634.715} C_VEL
LIN {X 0,Y 218.02,Z 349.39,A -85,B 0,C 180,E1 -21636.206,E2 -21636.206} C_VEL
LIN {X 0,Y 222.289,Z 356.156,A -85,B 0,C 180,E1 -21639.95,E2 -21639.95} C_VEL
LIN {X 0,Y 225.732,Z 361.916,A -85,B 0,C 180,E1 -21642.401,E2 -21642.401} C_VEL
LIN {X 0,Y 228.818,Z 367.506,A -85,B 0,C 180,E1 -21644.33,E2 -21644.33} C_VEL
LIN {X 0,Y 229.716,Z 369.2,A -85,B 0,C 180,E1 -21644.865,E2 -21644.865} C_VEL
LIN {X 0,Y 230.702,Z 372.019,A -85,B 0,C 180,E1 -21645.498,E2 -21645.498} C_VEL
LIN {X 0,Y 231.387,Z 377.999,A -85,B 0,C 180,E1 -21646.21,E2 -21646.21} C_VEL
LIN {X 0,Y 232.052,Z 385.519,A -85,B 0,C 180,E1 -21647.009,E2 -21647.009} C_VEL
LIN {X 0,Y 232.622,Z 387.704,A -85,B 0,C 180,E1 -21647.379,E2 -21647.379} C_VEL
LIN {X 0,Y 234.974,Z 394.483,A -85,B 0,C 180,E1 -21648.694,E2 -21648.694} C_VEL
LIN {X 0,Y 235.125,Z 398.743,A -85,B 0,C 180,E1 -21649.018,E2 -21649.018} C_VEL
LIN {X 0,Y 231.19,Z 441.323,A -85,B 0,C 180,E1 -21650.539,E2 -21650.539} C_VEL
LIN {X 0,Y 228.952,Z 454.979,A -85,B 0,C 180,E1 -21651.285,E2 -21651.285} C_VEL
LIN {X 0,Y 226.321,Z 466.494,A -85,B 0,C 180,E1 -21652.17,E2 -21652.17} C_VEL
LIN {X 0,Y 222.76,Z 478.754,A -85,B 0,C 180,E1 -21653.451,E2 -21653.451} C_VEL
LIN {X 0,Y 218.478,Z 491.058,A -85,B 0,C 180,E1 -21655.18,E2 -21655.18} C_VEL
LIN {X 0,Y 214.883,Z 499.939,A -85,B 0,C 180,E1 -21656.781,E2 -21656.781} C_VEL
LIN {X 0,Y 210.838,Z 509.217,A -85,B 0,C 180,E1 -21658.89,E2 -21658.89} C_VEL
LIN {X 0,Y 206.337,Z 518.279,A -85,B 0,C 180,E1 -21661.519,E2 -21661.519} C_VEL
LIN {X 0,Y 202.397,Z 525.649,A -85,B 0,C 180,E1 -21664.274,E2 -21664.274} C_VEL
LIN {X 0,Y 198.974,Z 531.624,A -85,B 0,C 180,E1 -21667.136,E2 -21667.136} C_VEL
LIN {X 0,Y 196.23,Z 536.408,A -85,B 0,C 180,E1 -21670.107,E2 -21670.107} C_VEL
LIN {X 0,Y 193.795,Z 540.138,A -85,B 0,C 180,E1 -21673.134,E2 -21673.134} C_VEL
LIN {X 0,Y 192.556,Z 542.093,A -85,B 0,C 180,E1 -21675.196,E2 -21675.196} C_VEL
LIN {X 0,Y 191.018,Z 544.704,A -85,B 0,C 180,E1 -21679.398,E2 -21679.398} C_VEL
LIN {X 0,Y 190.277,Z 545.776,A -85,B 0,C 180,E1 -21683.637,E2 -21683.637} C_VEL
LIN {X 0,Y 190.201,Z 545.652,A -85,B 0,C 180,E1 -21686.08,E2 -21686.08} C_VEL
LIN {X 0,Y 190.488,Z 544.344,A -85,B 0,C 180,E1 -21689.999,E2 -21689.999} C_VEL
LIN {X 0,Y 190.363,Z 543.025,A -85,B 0,C 180,E1 -21692.115,E2 -21692.115} C_VEL
LIN {X 0,Y 190.363,Z 540.887,A -85,B 0,C 180,E1 -21694.579,E2 -21694.579} C_VEL
LIN {X 0,Y 190.497,Z 537.651,A -85,B 0,C 180,E1 -21697.418,E2 -21697.418} C_VEL
LIN {X 0,Y 190.967,Z 532.884,A -85,B 0,C 180,E1 -21700.602,E2 -21700.602} C_VEL
LIN {X 0,Y 191.838,Z 526.793,A -85,B 0,C 180,E1 -21703.775,E2 -21703.775} C_VEL
LIN {X 0,Y 193.326,Z 519.189,A -85,B 0,C 180,E1 -21706.906,E2 -21706.906} C_VEL
LIN {X 0,Y 194.893,Z 511.4,A -85,B 0,C 180,E1 -21709.484,E2 -21709.484} C_VEL
LIN {X 0,Y 196.715,Z 502.326,A -85,B 0,C 180,E1 -21711.921,E2 -21711.921} C_VEL
LIN {X 0,Y 198.847,Z 491.352,A -85,B 0,C 180,E1 -21714.258,E2 -21714.258} C_VEL
LIN {X 0,Y 200.906,Z 479.703,A -85,B 0,C 180,E1 -21716.207,E2 -21716.207} C_VEL
LIN {X 0,Y 202.813,Z 467.474,A -85,B 0,C 180,E1 -21717.75,E2 -21717.75} C_VEL
LIN {X 0,Y 204.498,Z 454.266,A -85,B 0,C 180,E1 -21718.969,E2 -21718.969} C_VEL
LIN {X 0,Y 205.544,Z 442.429,A -85,B 0,C 180,E1 -21719.72,E2 -21719.72} C_VEL
LIN {X 0,Y 208.058,Z 390.192,A -85,B 0,C 180,E1 -21721.83,E2 -21721.83} C_VEL
LIN {X 0,Y 204.876,Z 363.299,A -85,B 0,C 180,E1 -21723.421,E2 -21723.421} C_VEL
LIN {X 0,Y 196.383,Z 339.767,A -85,B 0,C 180,E1 -21725.649,E2 -21725.649} C_VEL
LIN {X 0,Y 194.376,Z 334.232,A -85,B 0,C 180,E1 -21726.27,E2 -21726.27} C_VEL
LIN {X 0,Y 192.594,Z 326.498,A -85,B 0,C 180,E1 -21730.2,E2 -21730.2} C_VEL
LIN {X 0,Y 192.486,Z 326.506,A -85,B 0,C 180,E1 -21736.075,E2 -21736.075} C_VEL
LIN {X 0,Y 192.536,Z 326.503,A -85,B 0,C 180,E1 -21740.042,E2 -21740.042} C_VEL
LIN {X 0,Y 192.577,Z 326.496,A -85,B 0,C 180,E1 -21744.274,E2 -21744.274} C_VEL
LIN {X 0,Y 192.603,Z 326.469,A -85,B 0,C 180,E1 -21749.28,E2 -21749.28} C_VEL
LIN {X 0,Y 192.66,Z 326.479,A -85,B 0,C 180,E1 -21751.692,E2 -21751.692} C_VEL
LIN {X 0,Y 192.701,Z 326.482,A -85,B 0,C 180,E1 -21756.348,E2 -21756.348} C_VEL
LIN {X 0,Y 192.727,Z 326.477,A -85,B 0,C 180,E1 -21761.457,E2 -21761.457} C_VEL
LIN {X 0,Y 192.767,Z 326.473,A -85,B 0,C 180,E1 -21765.214,E2 -21765.214} C_VEL
LIN {X 0,Y 192.977,Z 326.439,A -85,B 0,C 180,E1 -21769.509,E2 -21769.509} C_VEL
LIN {X 0,Y 193.058,Z 326.437,A -85,B 0,C 180,E1 -21771.628,E2 -21771.628} C_VEL
LIN {X 0,Y 193.259,Z 326.398,A -85,B 0,C 180,E1 -21777.916,E2 -21777.916} C_VEL
LIN {X 0,Y 193.438,Z 326.377,A -85,B 0,C 180,E1 -21780,E2 -21780} C_VEL
LIN {X 0,Y 192.963,Z 326.446,A -85,B 0,C 180,E1 -21784.178,E2 -21784.178} C_VEL
LIN {X 0,Y 193.024,Z 326.431,A -85,B 0,C 180,E1 -21788.375,E2 -21788.375} C_VEL
LIN {X 0,Y 192.798,Z 326.453,A -85,B 0,C 180,E1 -21792.634,E2 -21792.634} C_VEL
LIN {X 0,Y 192.754,Z 326.47,A -85,B 0,C 180,E1 -21796.96,E2 -21796.96} C_VEL
LIN {X 0,Y 192.617,Z 326.484,A -85,B 0,C 180,E1 -21801.4,E2 -21801.4} C_VEL
LIN {X 0,Y 192.636,Z 326.471,A -85,B 0,C 180,E1 -21804.209,E2 -21804.209} C_VEL
LIN {X 0,Y 192.599,Z 326.488,A -85,B 0,C 180,E1 -21808.867,E2 -21808.867} C_VEL
LIN {X 0,Y 192.592,Z 326.494,A -85,B 0,C 180,E1 -21813.188,E2 -21813.188} C_VEL
LIN {X 0,Y 192.549,Z 326.488,A -85,B 0,C 180,E1 -21818.353,E2 -21818.353} C_VEL
LIN {X 0,Y 192.488,Z 326.502,A -85,B 0,C 180,E1 -21823.097,E2 -21823.097} C_VEL
LIN {X 0,Y 192.486,Z 326.509,A -85,B 0,C 180,E1 -21826.907,E2 -21826.907} C_VEL
LIN {X 0,Y 192.543,Z 326.487,A -85,B 0,C 180,E1 -21831.648,E2 -21831.648} C_VEL
LIN {X 0,Y 192.595,Z 326.492,A -85,B 0,C 180,E1 -21836.815,E2 -21836.815} C_VEL
LIN {X 0,Y 192.621,Z 326.491,A -85,B 0,C 180,E1 -21841.687,E2 -21841.687} C_VEL
LIN {X 0,Y 192.68,Z 326.482,A -85,B 0,C 180,E1 -21846.347,E2 -21846.347} C_VEL
LIN {X 0,Y 192.701,Z 326.481,A -85,B 0,C 180,E1 -21851.489,E2 -21851.489} C_VEL
LIN {X 0,Y 192.746,Z 326.474,A -85,B 0,C 180,E1 -21855.214,E2 -21855.214} C_VEL
LIN {X 0,Y 192.948,Z 326.451,A -85,B 0,C 180,E1 -21859.568,E2 -21859.568} C_VEL
LIN {X 0,Y 192.967,Z 326.449,A -85,B 0,C 180,E1 -21863.728,E2 -21863.728} C_VEL
LIN {X 0,Y 193.212,Z 326.419,A -85,B 0,C 180,E1 -21867.917,E2 -21867.917} C_VEL
LIN {X 0,Y 193.413,Z 326.395,A -85,B 0,C 180,E1 -21870.001,E2 -21870.001} C_VEL
LIN {X 0,Y 192.92,Z 326.457,A -85,B 0,C 180,E1 -21874.179,E2 -21874.179} C_VEL
LIN {X 0,Y 193.016,Z 326.443,A -85,B 0,C 180,E1 -21878.376,E2 -21878.376} C_VEL
LIN {X 0,Y 192.867,Z 326.461,A -85,B 0,C 180,E1 -21880.897,E2 -21880.897} C_VEL
LIN {X 0,Y 194.061,Z 329.641,A -85,B 0,C 180,E1 -21881.271,E2 -21881.271} C_VEL
LIN {X 0,Y 203.426,Z 350.662,A -85,B 0,C 180,E1 -21883.558,E2 -21883.558} C_VEL
LIN {X 0,Y 209.041,Z 366.894,A -85,B 0,C 180,E1 -21884.979,E2 -21884.979} C_VEL
LIN {X 0,Y 205.684,Z 429.358,A -85,B 0,C 180,E1 -21887.479,E2 -21887.479} C_VEL
LIN {X 0,Y 204.449,Z 442.883,A -85,B 0,C 180,E1 -21888.412,E2 -21888.412} C_VEL
LIN {X 0,Y 203.147,Z 454.612,A -85,B 0,C 180,E1 -21889.582,E2 -21889.582} C_VEL
LIN {X 0,Y 201.275,Z 467.056,A -85,B 0,C 180,E1 -21891.241,E2 -21891.241} C_VEL
LIN {X 0,Y 199.451,Z 477.875,A -85,B 0,C 180,E1 -21893.1,E2 -21893.1} C_VEL
LIN {X 0,Y 197.586,Z 487.964,A -85,B 0,C 180,E1 -21895.268,E2 -21895.268} C_VEL
LIN {X 0,Y 195.612,Z 497.543,A -85,B 0,C 180,E1 -21897.845,E2 -21897.845} C_VEL
LIN {X 0,Y 193.965,Z 505.472,A -85,B 0,C 180,E1 -21900.483,E2 -21900.483} C_VEL
LIN {X 0,Y 192.639,Z 512.087,A -85,B 0,C 180,E1 -21903.179,E2 -21903.179} C_VEL
LIN {X 0,Y 191.423,Z 518.986,A -85,B 0,C 180,E1 -21906.709,E2 -21906.709} C_VEL
LIN {X 0,Y 190.741,Z 522.951,A -85,B 0,C 180,E1 -21909.306,E2 -21909.306} C_VEL
LIN {X 0,Y 190.09,Z 526.594,A -85,B 0,C 180,E1 -21912.315,E2 -21912.315} C_VEL
LIN {X 0,Y 189.845,Z 529.274,A -85,B 0,C 180,E1 -21915.301,E2 -21915.301} C_VEL
LIN {X 0,Y 189.896,Z 531.082,A -85,B 0,C 180,E1 -21918.227,E2 -21918.227} C_VEL
LIN {X 0,Y 190.204,Z 532.067,A -85,B 0,C 180,E1 -21921.086,E2 -21921.086} C_VEL
LIN {X 0,Y 190.872,Z 532.316,A -85,B 0,C 180,E1 -21924.102,E2 -21924.102} C_VEL
LIN {X 0,Y 191.982,Z 531.687,A -85,B 0,C 180,E1 -21927.351,E2 -21927.351} C_VEL
LIN {X 0,Y 193.612,Z 530.076,A -85,B 0,C 180,E1 -21930.598,E2 -21930.598} C_VEL
LIN {X 0,Y 196.271,Z 526.692,A -85,B 0,C 180,E1 -21934.551,E2 -21934.551} C_VEL
LIN {X 0,Y 199.734,Z 521.69,A -85,B 0,C 180,E1 -21938.317,E2 -21938.317} C_VEL
LIN {X 0,Y 202.839,Z 516.786,A -85,B 0,C 180,E1 -21941.045,E2 -21941.045} C_VEL
LIN {X 0,Y 206.357,Z 510.653,A -85,B 0,C 180,E1 -21943.72,E2 -21943.72} C_VEL
LIN {X 0,Y 210.666,Z 502.445,A -85,B 0,C 180,E1 -21946.495,E2 -21946.495} C_VEL
LIN {X 0,Y 214.878,Z 493.347,A -85,B 0,C 180,E1 -21948.878,E2 -21948.878} C_VEL
LIN {X 0,Y 219.169,Z 482.902,A -85,B 0,C 180,E1 -21951.006,E2 -21951.006} C_VEL
LIN {X 0,Y 223.093,Z 471.785,A -85,B 0,C 180,E1 -21952.76,E2 -21952.76} C_VEL
LIN {X 0,Y 226.742,Z 458.898,A -85,B 0,C 180,E1 -21954.301,E2 -21954.301} C_VEL
LIN {X 0,Y 229.355,Z 446.916,A -85,B 0,C 180,E1 -21955.386,E2 -21955.386} C_VEL
LIN {X 0,Y 231.357,Z 434.957,A -85,B 0,C 180,E1 -21956.135,E2 -21956.135} C_VEL
LIN {X 0,Y 232.933,Z 420.094,A -85,B 0,C 180,E1 -21956.742,E2 -21956.742} C_VEL
LIN {X 0,Y 235.913,Z 386.395,A -85,B 0,C 180,E1 -21957.943,E2 -21957.943} C_VEL
LIN {X 0,Y 231.826,Z 377.236,A -85,B 0,C 180,E1 -21960.092,E2 -21960.092} C_VEL
LIN {X 0,Y 226.344,Z 367.141,A -85,B 0,C 180,E1 -21963.274,E2 -21963.274} C_VEL
LIN {X 0,Y 223.661,Z 363.103,A -85,B 0,C 180,E1 -21964.996,E2 -21964.996} C_VEL
LIN {X 0,Y 221.424,Z 360.042,A -85,B 0,C 180,E1 -21966.592,E2 -21966.592} C_VEL
LIN {X 0,Y 218.733,Z 356.595,A -85,B 0,C 180,E1 -21968.744,E2 -21968.744} C_VEL
LIN {X 0,Y 217.83,Z 355.079,A -85,B 0,C 180,E1 -21969.615,E2 -21969.615} C_VEL
LIN {X 0,Y 215.358,Z 352.184,A -85,B 0,C 180,E1 -21972.142,E2 -21972.142} C_VEL
LIN {X 0,Y 214.379,Z 350.568,A -85,B 0,C 180,E1 -21973.454,E2 -21973.454} C_VEL
LIN {X 0,Y 211.021,Z 347.123,A -85,B 0,C 180,E1 -21980.214,E2 -21980.214} C_VEL
LIN {X 0,Y 210.639,Z 347.032,A -85,B 0,C 180,E1 -21983.602,E2 -21983.602} C_VEL
LIN {X 0,Y 211.552,Z 348.275,A -85,B 0,C 180,E1 -21988.214,E2 -21988.214} C_VEL
LIN {X 0,Y 215.213,Z 354.535,A -85,B 0,C 180,E1 -21994.528,E2 -21994.528} C_VEL
LIN {X 0,Y 216.436,Z 356.369,A -85,B 0,C 180,E1 -21995.868,E2 -21995.868} C_VEL
LIN {X 0,Y 220.01,Z 362.206,A -85,B 0,C 180,E1 -21999.19,E2 -21999.19} C_VEL
LIN {X 0,Y 223.34,Z 368.129,A -85,B 0,C 180,E1 -22001.739,E2 -22001.739} C_VEL
LIN {X 0,Y 226.115,Z 373.382,A -85,B 0,C 180,E1 -22003.571,E2 -22003.571} C_VEL
LIN {X 0,Y 228.283,Z 377.777,A -85,B 0,C 180,E1 -22004.919,E2 -22004.919} C_VEL
LIN {X 0,Y 231.409,Z 384.728,A -85,B 0,C 180,E1 -22006.708,E2 -22006.708} C_VEL
LIN {X 0,Y 232.622,Z 387.704,A -85,B 0,C 180,E1 -22007.379,E2 -22007.379} C_VEL
LIN {X 0,Y 233.296,Z 390.951,A -85,B 0,C 180,E1 -22007.855,E2 -22007.855} C_VEL
LIN {X 0,Y 233.337,Z 395.617,A -85,B 0,C 180,E1 -22008.192,E2 -22008.192} C_VEL
LIN {X 0,Y 232.403,Z 402.494,A -85,B 0,C 180,E1 -22008.33,E2 -22008.33} C_VEL
LIN {X 0,Y 229.437,Z 417.13,A -85,B 0,C 180,E1 -22008.27,E2 -22008.27} C_VEL
LIN {X 0,Y 229.169,Z 419.232,A -85,B 0,C 180,E1 -22008.32,E2 -22008.32} C_VEL
LIN {X 0,Y 226.752,Z 442.25,A -85,B 0,C 180,E1 -22009.17,E2 -22009.17} C_VEL
LIN {X 0,Y 224.413,Z 455.469,A -85,B 0,C 180,E1 -22009.911,E2 -22009.911} C_VEL
LIN {X 0,Y 221.413,Z 467.734,A -85,B 0,C 180,E1 -22010.885,E2 -22010.885} C_VEL
LIN {X 0,Y 217.729,Z 479.658,A -85,B 0,C 180,E1 -22012.171,E2 -22012.171} C_VEL
LIN {X 0,Y 213.291,Z 491.729,A -85,B 0,C 180,E1 -22013.914,E2 -22013.914} C_VEL
LIN {X 0,Y 209.109,Z 501.424,A -85,B 0,C 180,E1 -22015.738,E2 -22015.738} C_VEL
LIN {X 0,Y 204.049,Z 511.927,A -85,B 0,C 180,E1 -22018.314,E2 -22018.314} C_VEL
LIN {X 0,Y 199.481,Z 520.406,A -85,B 0,C 180,E1 -22021.024,E2 -22021.024} C_VEL
LIN {X 0,Y 195.402,Z 527.314,A -85,B 0,C 180,E1 -22023.857,E2 -22023.857} C_VEL
LIN {X 0,Y 191.489,Z 533.719,A -85,B 0,C 180,E1 -22027.332,E2 -22027.332} C_VEL
LIN {X 0,Y 188.653,Z 537.979,A -85,B 0,C 180,E1 -22030.409,E2 -22030.409} C_VEL
LIN {X 0,Y 187.019,Z 540.273,A -85,B 0,C 180,E1 -22032.503,E2 -22032.503} C_VEL
LIN {X 0,Y 185.67,Z 542.106,A -85,B 0,C 180,E1 -22034.634,E2 -22034.634} C_VEL
LIN {X 0,Y 184.03,Z 544.584,A -85,B 0,C 180,E1 -22038.991,E2 -22038.991} C_VEL
LIN {X 0,Y 183.502,Z 545.25,A -85,B 0,C 180,E1 -22041.187,E2 -22041.187} C_VEL
LIN {X 0,Y 183.21,Z 545.504,A -85,B 0,C 180,E1 -22043.39,E2 -22043.39} C_VEL
LIN {X 0,Y 183.218,Z 544.811,A -85,B 0,C 180,E1 -22047.8,E2 -22047.8} C_VEL
LIN {X 0,Y 183.424,Z 543.878,A -85,B 0,C 180,E1 -22049.999,E2 -22049.999} C_VEL
LIN {X 0,Y 183.285,Z 542.479,A -85,B 0,C 180,E1 -22052.196,E2 -22052.196} C_VEL
LIN {X 0,Y 183.311,Z 539.506,A -85,B 0,C 180,E1 -22055.498,E2 -22055.498} C_VEL
LIN {X 0,Y 183.577,Z 535.405,A -85,B 0,C 180,E1 -22058.807,E2 -22058.807} C_VEL
LIN {X 0,Y 184.385,Z 529.03,A -85,B 0,C 180,E1 -22062.659,E2 -22062.659} C_VEL
LIN {X 0,Y 185.652,Z 522.052,A -85,B 0,C 180,E1 -22065.928,E2 -22065.928} C_VEL
LIN {X 0,Y 187.08,Z 514.897,A -85,B 0,C 180,E1 -22068.62,E2 -22068.62} C_VEL
LIN {X 0,Y 188.956,Z 505.852,A -85,B 0,C 180,E1 -22071.372,E2 -22071.372} C_VEL
LIN {X 0,Y 191.01,Z 495.528,A -85,B 0,C 180,E1 -22073.873,E2 -22073.873} C_VEL
LIN {X 0,Y 193.077,Z 484.989,A -85,B 0,C 180,E1 -22075.898,E2 -22075.898} C_VEL
LIN {X 0,Y 195.177,Z 473.46,A -85,B 0,C 180,E1 -22077.619,E2 -22077.619} C_VEL
LIN {X 0,Y 197.011,Z 460.422,A -85,B 0,C 180,E1 -22079.079,E2 -22079.079} C_VEL
LIN {X 0,Y 198.49,Z 447.714,A -85,B 0,C 180,E1 -22080.08,E2 -22080.08} C_VEL
LIN {X 0,Y 199.446,Z 431.641,A -85,B 0,C 180,E1 -22080.872,E2 -22080.872} C_VEL
LIN {X 0,Y 201.439,Z 390.736,A -85,B 0,C 180,E1 -22082.554,E2 -22082.554} C_VEL
LIN {X 0,Y 198.544,Z 365.411,A -85,B 0,C 180,E1 -22084.111,E2 -22084.111} C_VEL
LIN {X 0,Y 189.546,Z 340.509,A -85,B 0,C 180,E1 -22086.592,E2 -22086.592} C_VEL
LIN {X 0,Y 187.088,Z 334.044,A -85,B 0,C 180,E1 -22087.313,E2 -22087.313} C_VEL
LIN {X 0,Y 185.533,Z 327.375,A -85,B 0,C 180,E1 -22090.94,E2 -22090.94} C_VEL
LIN {X 0,Y 185.455,Z 327.382,A -85,B 0,C 180,E1 -22096.054,E2 -22096.054} C_VEL
LIN {X 0,Y 185.485,Z 327.381,A -85,B 0,C 180,E1 -22099.9,E2 -22099.9} C_VEL
LIN {X 0,Y 185.54,Z 327.373,A -85,B 0,C 180,E1 -22102.695,E2 -22102.695} C_VEL
LIN {X 0,Y 185.541,Z 327.36,A -85,B 0,C 180,E1 -22107.975,E2 -22107.975} C_VEL
LIN {X 0,Y 185.578,Z 327.347,A -85,B 0,C 180,E1 -22110.575,E2 -22110.575} C_VEL
LIN {X 0,Y 185.583,Z 327.371,A -85,B 0,C 180,E1 -22115.382,E2 -22115.382} C_VEL
LIN {X 0,Y 185.67,Z 327.354,A -85,B 0,C 180,E1 -22121.133,E2 -22121.133} C_VEL
LIN {X 0,Y 185.72,Z 327.35,A -85,B 0,C 180,E1 -22124.64,E2 -22124.64} C_VEL
LIN {X 0,Y 185.92,Z 327.317,A -85,B 0,C 180,E1 -22129.359,E2 -22129.359} C_VEL
LIN {X 0,Y 185.957,Z 327.323,A -85,B 0,C 180,E1 -22133.49,E2 -22133.49} C_VEL
LIN {X 0,Y 186.203,Z 327.277,A -85,B 0,C 180,E1 -22137.837,E2 -22137.837} C_VEL
LIN {X 0,Y 186.402,Z 327.252,A -85,B 0,C 180,E1 -22140.001,E2 -22140.001} C_VEL
LIN {X 0,Y 185.91,Z 327.324,A -85,B 0,C 180,E1 -22144.337,E2 -22144.337} C_VEL
LIN {X 0,Y 185.973,Z 327.308,A -85,B 0,C 180,E1 -22148.695,E2 -22148.695} C_VEL
LIN {X 0,Y 185.725,Z 327.334,A -85,B 0,C 180,E1 -22153.124,E2 -22153.124} C_VEL
LIN {X 0,Y 185.686,Z 327.35,A -85,B 0,C 180,E1 -22157.626,E2 -22157.626} C_VEL
LIN {X 0,Y 185.574,Z 327.359,A -85,B 0,C 180,E1 -22162.255,E2 -22162.255} C_VEL
LIN {X 0,Y 185.505,Z 327.362,A -85,B 0,C 180,E1 -22167.042,E2 -22167.042} C_VEL
LIN {X 0,Y 185.541,Z 327.367,A -85,B 0,C 180,E1 -22169.501,E2 -22169.501} C_VEL
LIN {X 0,Y 185.495,Z 327.378,A -85,B 0,C 180,E1 -22174.634,E2 -22174.634} C_VEL
LIN {X 0,Y 185.503,Z 327.367,A -85,B 0,C 180,E1 -22177.315,E2 -22177.315} C_VEL
LIN {X 0,Y 185.468,Z 327.363,A -85,B 0,C 180,E1 -22180.726,E2 -22180.726} C_VEL
LIN {X 0,Y 185.456,Z 327.382,A -85,B 0,C 180,E1 -22186.057,E2 -22186.057} C_VEL
LIN {X 0,Y 185.458,Z 327.377,A -85,B 0,C 180,E1 -22189.895,E2 -22189.895} C_VEL
LIN {X 0,Y 185.501,Z 327.363,A -85,B 0,C 180,E1 -22192.715,E2 -22192.715} C_VEL
LIN {X 0,Y 185.531,Z 327.373,A -85,B 0,C 180,E1 -22197.974,E2 -22197.974} C_VEL
LIN {X 0,Y 185.547,Z 327.369,A -85,B 0,C 180,E1 -22200.597,E2 -22200.597} C_VEL
LIN {X 0,Y 185.581,Z 327.367,A -85,B 0,C 180,E1 -22205.383,E2 -22205.383} C_VEL
LIN {X 0,Y 185.636,Z 327.359,A -85,B 0,C 180,E1 -22211.172,E2 -22211.172} C_VEL
LIN {X 0,Y 185.674,Z 327.354,A -85,B 0,C 180,E1 -22214.637,E2 -22214.637} C_VEL
LIN {X 0,Y 185.891,Z 327.329,A -85,B 0,C 180,E1 -22219.42,E2 -22219.42} C_VEL
